// TwinCAT 3 PLC project MONETSRuntime
// Title: MONETS
// Company: IAG
// ProjectVersion: 1.2.0
// ProgramVersion: 3.1.4026.13
// libraries:
//   AstroBROT, * (BROT)
//   BROTLib, * (BROT)
//   HalfBROT, * (BROT)
//   MONET Roof, * (Georg-August-Universitaet Goettingen)
//   MONETcommon, * (IAG)
//   Tc2_DataExchange, * (Beckhoff Automation GmbH)
//   Tc2_Math, * (Beckhoff Automation GmbH)
//   Tc2_MC2, * (Beckhoff Automation GmbH)
//   Tc2_MC2_Drive, * (Beckhoff Automation GmbH)
//   Tc2_NC, * (Beckhoff Automation GmbH)
//   Tc2_Standard, * (Beckhoff Automation GmbH)
//   Tc2_System, * (Beckhoff Automation GmbH)
//   Tc2_Utilities, * (Beckhoff Automation GmbH)
//   Tc3_IotBase, * (Beckhoff Automation GmbH)
//   Tc3_JsonXml, * (Beckhoff Automation GmbH)
//   Tc3_Module, * (Beckhoff Automation GmbH)
//   VisuDialogs, * (System)
//   VisuElemEventTable, * (System)
//   VisuSymbols,3.5.10.0,System
// project tree:
//   / GlobalTextList.TcGTLO, PlcTask.TcTTO (not stored), VisualizationManager.TcVMO (not stored)
//   POUs/ FB_TelescopeAuxiliary.TcPOU, FB_WeatherCheck.TcPOU, MAIN.TcPOU
//   VISUs/ Azimuth.TcVIS, Cover.TcVIS, Derotator.TcVIS, Elevation.TcVIS, Focus.TcVIS, Hydraulics.TcVIS, Pendant.TcVIS, Safety.TcVIS, Telescope.TcVIS, Visualization.TcVIS, Roof.TcVIS
//   GVLs/ Global_Version.TcGVL
// real-time tasks:
//   TASK PlcTask: cycle T#10ms, priority 20, ADS port 350
// motion (NC):
//   TASK NC-Task 1 SAF: cycle T#2ms, priority 4, ADS port 501
//   TASK NC-Task 1 SVB: cycle T#10ms, priority 8, ADS port 511
//   AXIS Azimuth (id 1)
//     General: UnitName=°
//     Dynamic: AccelerationMaximum=10, DecelerationMaximum=10, Acceleration=3, Deceleration=3, Jerk=1
//     Velo: RefSearch=2, RefSync=2, SlowManual=1, FastManual=5, Fast=684, Maximum=10
//     OtherSettings: AllowMotionCmdToSlave=true
//     encoder EncType=8
//       EncPara: ScaleFactorNumerator=360, ScaleFactorDenominator=1048576, MaxCount=#xffffffff
//         SoftEndMinControl: Enable=true, Range=-274
//         SoftEndMaxControl: Enable=true, Range=270
//         Inc: RefMode=2
//     drive DrvType=9
//       DrvPara: MaxCount=#xffffffff, DriveControlDWord=#x00030100
//         Analog: VeloReferenz=752.4, VeloScale=1.02400649589962, TorqueSetpointScale=10, ScaleFactorActTorque=0.1
//         TimeComp: TaskDelayCycles=1
//     controller CtrType=1
//       CtrPara: PriorControlFactor=1
//         PosDiffControl: Range=10
//         Observer: BandWidth=20
//   AXIS Elevation (id 2)
//     General: UnitName=°
//     Dynamic: AccelerationMaximum=10, DecelerationMaximum=10, Acceleration=3, Deceleration=3, Jerk=2
//     Velo: RefSearch=1, RefSync=2, SlowManual=1, FastManual=3, Fast=1425, Maximum=10
//     OtherSettings: AllowMotionCmdToSlave=true
//     encoder EncType=8
//       EncPara: ScaleFactorNumerator=360, ScaleFactorDenominator=1048576, MaxCount=#xffffffff
//         SoftEndMinControl: Enable=true
//         SoftEndMaxControl: Enable=true, Range=91
//         Inc: RefMode=2
//     drive DrvType=9
//       DrvPara: MaxCount=#xffffffff, DriveControlDWord=#x00030100
//         Analog: VeloReferenz=1567.5, VeloScale=1.02400649589962, TorqueSetpointScale=10, ScaleFactorActTorque=0.1
//         TimeComp: TaskDelayCycles=1
//     controller CtrType=1
//       CtrPara: PriorControlFactor=1
//         Observer: BandWidth=20
//   AXIS Derotator (id 3)
//     General: UnitName=°
//     Dynamic: AccelerationMaximum=20, DecelerationMaximum=20, Acceleration=17.5833776855469, Deceleration=17.5833776855469, Jerk=52.7501330566406
//     Velo: RefSearch=1, RefSync=0.5, SlowManual=0.5, FastManual=5, Fast=11.7222517903646, Maximum=11.7222517903646
//     OtherSettings: AllowMotionCmdToSlave=true
//     encoder EncType=8
//       EncPara: ScaleFactorNumerator=0.2, ScaleFactorDenominator=1048576, Offset=255.939444732666, MaxCount=#xffffffff, ReferenceSystem=1
//         SoftEndMinControl: Enable=true, Range=-90
//         SoftEndMaxControl: Enable=true, Range=360
//     drive DrvType=9
//       DrvPara: MaxCount=#xffffffff, DriveControlDWord=#x00030100
//         Analog: VeloReferenz=12.894476969401, VeloScale=1.02400649589962, TorqueSetpointScale=10, ScaleFactorActTorque=0.1
//         TimeComp: TaskDelayCycles=1
//     controller CtrType=1
//       CtrPara: PriorControlFactor=1
//         Observer: BandWidth=20
//   AXIS Focus (id 4)
//     Dynamic: AccelerationMaximum=100, DecelerationMaximum=100, Acceleration=4.5, Deceleration=4.5, Jerk=13.5
//     Velo: RefSearch=0.2, RefSync=0.2, SlowManual=0.1, FastManual=0.5, Maximum=5
//     OtherSettings: AllowMotionCmdToSlave=true, PulseDistancePos=1, PulseDistanceNeg=1
//     encoder EncType=4
//       EncPara: ScaleFactorNumerator=0.001, ScaleFactorDenominator=5, Inverse=true, MaxCount=#x0000ffff
//         SoftEndMaxControl: Range=100
//         Inc: RefMode=2, RefSoftSyncMask=#x0000ffff
//     drive DrvType=23
//       DrvPara: Inverse=true
//         Analog: VeloReferenz=10.27313178, TorqueSetpointScale=10, ScaleFactorActTorque=0.1
//         TimeComp: TaskDelayCycles=1
//     controller CtrType=1
//       CtrPara: PriorControlFactor=1
//         PID: PosKp=200
//         Observer: BandWidth=20
// I/O:
//   DEVICE Device 1 (EtherCAT), AmsNetId 0.0.0.0.2.1
//     Term 8 (EK1200) [EK1200-5000 EtherCAT Power supply (2A E-Bus)]
//       Term 25 (EL1004) [EL1004 4Ch. Dig. Input 24V, 3ms]
//       Temperature IN (EL3202) [EL3202 2Ch. Ana. Input PT100 (RTD)]
//       Brake AzEl (EL2004) [EL2004 4Ch. Dig. Output 24V, 0.5A]
//       Safety Logic (EL6910) [EL6910, TwinSAFE PLC]
//       Safety IN (EL1904) [EL1904, 4 Ch. Safety Input 24V, TwinSAFE]
//         modules: Module 1 (FSOES)
//       Safety OUT (EL2904) [EL2904, 4 Ch. Safety Output 24V, 0.5A, TwinSAFE]
//         modules: Module 1 (FSOES), Module 2 (DO)
//       Hydraulics OUT (EL2008) [EL2008 8Ch. Dig. Output 24V, 0.5A]
//       Hydraulics Focus IN (EL1008) [EL1008 8Ch. Dig. Input 24V, 3ms]
//       Hydraulics IN2 (EL1008) [EL1008 8Ch. Dig. Input 24V, 3ms]
//       Focus Encoder (EL5101-0010) [EL5101-0010 1Ch. Inc. Encoder 5V (20 million increments/s)]
//       Focus Motor (EL7342) [EL7342 2Ch. DC motor output stage (50V, 3.5A)]
//       Mirror Temperature IN (EL3164) [EL3164 4Ch. Ana. Input 0-10V]
//       Power Analysis (EL3483) [EL3483 3Ch. Mains Monitoring]
//       Power (EL9410) [EL9410 E-Bus Power Supplier  (Diagnostics)]
//       Mirror Cover OUT1 (EL2004) [EL2004 4Ch. Dig. Output 24V, 0.5A]
//       Mirror Cover OUT2 (EL2004) [EL2004 4Ch. Dig. Output 24V, 0.5A]
//       Mirror Cover IN (EL1008) [EL1008 8Ch. Dig. Input 24V, 3ms]
//       Front Panel IN (EL1008) [EL1008 8Ch. Dig. Input 24V, 3ms]
//       Front Panel OUT (EL2004) [EL2004 4Ch. Dig. Output 24V, 0.5A]
//       Pendant Control IN (EL1008) [EL1008 8Ch. Dig. Input 24V, 3ms]
//       Pendant Control IN2 (EL1008) [EL1008 8Ch. Dig. Input 24V, 3ms]
//       Pendant Control OUT (EL2008) [EL2008 8Ch. Dig. Output 24V, 0.5A]
//       Cabinet OUT (EL2004) [EL2004 4Ch. Dig. Output 24V, 0.5A]
//       Term 32 (EL9011) [EL9011 End Terminal]
//   DEVICE Device 4 (EtherCAT), AmsNetId 0.0.0.0.5.1
//     Azimuth (AX5125-0000-0214) [AX5125-0000-0214 EtherCAT Drive (SoE, 1 Ch.)]
//       Term 9 (AX5805) [AX5805 (Safety Drive Option)]
//         modules: Module 1 (Safety Process Data, 1 axis), Module 2 (Standard Process Data, 1 axis)
//     Elevation (AX5125-0000-0214) [AX5125-0000-0214 EtherCAT Drive (SoE, 1 Ch.)]
//       Term 11 (AX5805) [AX5805 (Safety Drive Option)]
//         modules: Module 1 (Safety Process Data, 1 axis), Module 2 (Standard Process Data, 1 axis)
//     Derotator (AX5206-0000-0215) [AX5206-0000-0215 EtherCAT Drive (SoE, 2 Ch.)]
//       Term 13 (AX5805) [AX5805 (Safety Drive Option)]
//         modules: Module 1 (Safety Process Data, 2 axis), Module 2 (Standard Process Data, 2 axis)
//     Term 11 (EK1100) [EK1100 EtherCAT Coupler (2A E-Bus)]
//       Roof Open/Close (EL2008) [EL2008 8Ch. Dig. Output 24V, 0.5A]
//       Roof Reset (EL2008) [EL2008 8Ch. Dig. Output 24V, 0.5A]
//       Roof Safety OUT (EL2904) [EL2904, 4 Ch. Safety Output 24V, 0.5A, TwinSAFE]
//         modules: Module 1 (FSOES), Module 2 (DO)
//       Roof Safety IN (EL1904) [EL1904, 4 Ch. Safety Input 24V, TwinSAFE]
//         modules: Module 1 (FSOES)
//       Roof IN 1 (EL1008) [EL1008 8Ch. Dig. Input 24V, 3ms]
//       Roof IN 2 (EL1008) [EL1008 8Ch. Dig. Input 24V, 3ms]
//       Roof IN 3 (EL1008) [EL1008 8Ch. Dig. Input 24V, 3ms]
//       Roof Speed (EL4004) [EL4004 4Ch. Ana. Output 0-10V, 12bit]
//       Term 16 (EL9011) [EL9011 End Terminal]
// variable links:
//   Device 1 (EtherCAT) <-> Device 1 (EtherCAT)/Term 8 (EK1200)/Safety IN (EL1904)
//     Term 8 (EK1200)/Safety Logic (EL6910)/ConnectionInputs/Message_7 TxPDO <-> Module 1 (FSOES)/RxPDO/FSOE
//   Device 1 (EtherCAT) <-> Device 1 (EtherCAT)/Term 8 (EK1200)/Safety Logic (EL6910)
//     Term 8 (EK1200)/Safety IN (EL1904)/Module 1 (FSOES)/TxPDO/FSOE <-> ConnectionOutputs/Message_7 RxPDO
//     Term 8 (EK1200)/Safety OUT (EL2904)/Module 1 (FSOES)/RxPDO/FSOE <-> ConnectionInputs/Message_8 TxPDO
//   Device 1 (EtherCAT) <-> Device 1 (EtherCAT)/Term 8 (EK1200)/Safety OUT (EL2904)
//     Term 8 (EK1200)/Safety Logic (EL6910)/ConnectionOutputs/Message_8 RxPDO <-> Module 1 (FSOES)/TxPDO/FSOE
//   Device 1 (EtherCAT) <-> Device 4 (EtherCAT)/Azimuth (AX5125-0000-0214)/Term 9 (AX5805)
//     Term 8 (EK1200)/Safety Logic (EL6910)/ConnectionInputs/Message_5 TxPDO <-> Module 1 (Safety Process Data, 1 axis)/Outputs (Controlword)/FSOE
//   Device 1 (EtherCAT) <-> Device 4 (EtherCAT)/Derotator (AX5206-0000-0215)/Term 13 (AX5805)
//     Term 8 (EK1200)/Safety Logic (EL6910)/ConnectionInputs/Message_17 TxPDO <-> Module 1 (Safety Process Data, 2 axis)/Outputs (Controlword)/FSOE
//   Device 1 (EtherCAT) <-> Device 4 (EtherCAT)/Elevation (AX5125-0000-0214)/Term 11 (AX5805)
//     Term 8 (EK1200)/Safety Logic (EL6910)/ConnectionOutputs/Message_6 RxPDO <-> Module 1 (Safety Process Data, 1 axis)/Inputs (Statusword)/FSOE
//   Device 1 (EtherCAT) <-> Device 4 (EtherCAT)/Term 11 (EK1100)/Roof Safety IN (EL1904)
//     Term 8 (EK1200)/Safety Logic (EL6910)/ConnectionInputs/Message_29 TxPDO <-> Module 1 (FSOES)/RxPDO/FSOE
//   Device 1 (EtherCAT) <-> Device 4 (EtherCAT)/Term 11 (EK1100)/Roof Safety OUT (EL2904)
//     Term 8 (EK1200)/Safety Logic (EL6910)/ConnectionOutputs/Message_30 RxPDO <-> Module 1 (FSOES)/TxPDO/FSOE
//   Device 4 (EtherCAT) <-> Device 1 (EtherCAT)/Term 8 (EK1200)/Safety Logic (EL6910)
//     Azimuth (AX5125-0000-0214)/Term 9 (AX5805)/Module 1 (Safety Process Data, 1 axis)/Inputs (Statusword)/FSOE <-> ConnectionOutputs/Message_5 RxPDO
//     Derotator (AX5206-0000-0215)/Term 13 (AX5805)/Module 1 (Safety Process Data, 2 axis)/Inputs (Statusword)/FSOE <-> ConnectionOutputs/Message_17 RxPDO
//     Elevation (AX5125-0000-0214)/Term 11 (AX5805)/Module 1 (Safety Process Data, 1 axis)/Outputs (Controlword)/FSOE <-> ConnectionInputs/Message_6 TxPDO
//     Term 11 (EK1100)/Roof Safety IN (EL1904)/Module 1 (FSOES)/TxPDO/FSOE <-> ConnectionOutputs/Message_29 RxPDO
//     Term 11 (EK1100)/Roof Safety OUT (EL2904)/Module 1 (FSOES)/RxPDO/FSOE <-> ConnectionInputs/Message_30 TxPDO
//   NC-Task 1 SAF/Axes/Azimuth <-> Device 4 (EtherCAT)/Azimuth (AX5125-0000-0214)
//     Drive/Inputs/In/nDataIn1 <-> AT/Following distance
//     Drive/Inputs/In/nDataIn3[0] <-> AT/Torque/force feedback value
//     Drive/Inputs/In/nDcOutputTime <-> InfoData/DcOutputShift
//     Drive/Inputs/In/nState1 <-> AT/Drive status word @bit 8
//     Drive/Inputs/In/nState2 <-> AT/Drive status word
//     Drive/Inputs/In/nState4 @bit 1 <-> WcState/InputToggle
//     Drive/Inputs/In/nState4 <-> WcState/WcState
//     Drive/Outputs/Out/nCtrl1 <-> MDT/Master control word @bit 8
//     Drive/Outputs/Out/nDataOut1 <-> MDT/Position command value
//     Enc/Inputs/In/nDataIn1 <-> AT/Position feedback 1 value
//     Enc/Inputs/In/nDataIn3 <-> AT/Probe value 1 positive edge
//     Enc/Inputs/In/nDataIn7 <-> AT/Velocity feedback 1 value
//     Enc/Inputs/In/nDcInputTime <-> InfoData/DcInputShift
//     Enc/Inputs/In/nState4 @bit 1 <-> WcState/InputToggle
//     Enc/Inputs/In/nState4 <-> WcState/WcState
//     Enc/Inputs/In/nState5 <-> AT/Probe 1 positive latched
//     Enc/Outputs/Out/nCtrl5 <-> MDT/Probe 1 enable
//   NC-Task 1 SAF/Axes/Derotator <-> Device 4 (EtherCAT)/Derotator (AX5206-0000-0215)
//     Drive/Inputs/In/nDataIn1 <-> AT 2/Following distance
//     Drive/Inputs/In/nDataIn3[0] <-> AT 2/Torque/force feedback value
//     Drive/Inputs/In/nDcOutputTime <-> InfoData/DcOutputShift
//     Drive/Inputs/In/nState1 <-> AT 2/Drive status word @bit 8
//     Drive/Inputs/In/nState2 <-> AT 2/Drive status word
//     Drive/Inputs/In/nState4 @bit 1 <-> WcState/InputToggle
//     Drive/Inputs/In/nState4 <-> WcState/WcState
//     Drive/Outputs/Out/nCtrl1 <-> MDT 2/Master control word @bit 8
//     Drive/Outputs/Out/nDataOut1 <-> MDT 2/Position command value
//     Enc/Inputs/In/nDataIn1 <-> AT 2/Position feedback 1 value
//     Enc/Inputs/In/nDataIn7 <-> AT 2/Velocity feedback 1 value
//     Enc/Inputs/In/nDcInputTime <-> InfoData/DcInputShift
//     Enc/Inputs/In/nState4 @bit 1 <-> WcState/InputToggle
//     Enc/Inputs/In/nState4 <-> WcState/WcState
//   NC-Task 1 SAF/Axes/Elevation <-> Device 4 (EtherCAT)/Elevation (AX5125-0000-0214)
//     Drive/Inputs/In/nDataIn1 <-> AT/Following distance
//     Drive/Inputs/In/nDataIn3[0] <-> AT/Torque/force feedback value
//     Drive/Inputs/In/nDcOutputTime <-> InfoData/DcOutputShift
//     Drive/Inputs/In/nState1 <-> AT/Drive status word @bit 8
//     Drive/Inputs/In/nState2 <-> AT/Drive status word
//     Drive/Inputs/In/nState4 @bit 1 <-> WcState/InputToggle
//     Drive/Inputs/In/nState4 <-> WcState/WcState
//     Drive/Outputs/Out/nCtrl1 <-> MDT/Master control word @bit 8
//     Drive/Outputs/Out/nDataOut1 <-> MDT/Position command value
//     Enc/Inputs/In/nDataIn1 <-> AT/Position feedback 1 value
//     Enc/Inputs/In/nDataIn3 <-> AT/Probe value 1 positive edge
//     Enc/Inputs/In/nDataIn7 <-> AT/Velocity feedback 1 value
//     Enc/Inputs/In/nDcInputTime <-> InfoData/DcInputShift
//     Enc/Inputs/In/nState4 @bit 1 <-> WcState/InputToggle
//     Enc/Inputs/In/nState4 <-> WcState/WcState
//     Enc/Inputs/In/nState5 <-> AT/Probe 1 positive latched
//     Enc/Outputs/Out/nCtrl5 <-> MDT/Probe 1 enable
//   NC-Task 1 SAF/Axes/Focus <-> Device 1 (EtherCAT)/Term 8 (EK1200)/Focus Encoder (EL5101-0010)
//     Enc/Inputs/In/nDataIn1[0] <-> ENC Status compact/Counter value
//     Enc/Inputs/In/nDataIn2[0] <-> ENC Status compact/Latch value
//     Enc/Inputs/In/nState1 <-> ENC Status compact/Status/Latch C valid
//     Enc/Inputs/In/nState1 @bit 1 <-> ENC Status compact/Status/Latch extern valid
//     Enc/Inputs/In/nState1 @bit 6 <-> ENC Status compact/Status/Open circuit
//     Enc/Inputs/In/nState1 @bit 2 <-> ENC Status compact/Status/Set counter done
//     Enc/Inputs/In/nState1 @bit 5 <-> ENC Status compact/Status/Status of input status
//     Enc/Inputs/In/nState2 @bit 4 <-> ENC Status compact/Status/Status of extern latch
//     Enc/Inputs/In/nState2 <-> ENC Status compact/Status/Status of input A
//     Enc/Inputs/In/nState2 @bit 1 <-> ENC Status compact/Status/Status of input B
//     Enc/Inputs/In/nState2 @bit 2 <-> ENC Status compact/Status/Status of input C
//     Enc/Inputs/In/nState2 @bit 3 <-> ENC Status compact/Status/Status of input gate
//     Enc/Inputs/In/nState2 @bit 5 <-> ENC Status compact/Status/Sync error
//     Enc/Inputs/In/nState2 @bit 6 <-> ENC Status compact/Status/TxPDO State
//     Enc/Inputs/In/nState2 @bit 7 <-> ENC Status compact/Status/TxPDO Toggle
//     Enc/Inputs/In/nState4 @bit 1 <-> WcState/InputToggle
//     Enc/Inputs/In/nState4 <-> WcState/WcState
//     Enc/Outputs/Out/nCtrl1 <-> ENC Control compact/Control/Enable latch C
//     Enc/Outputs/Out/nCtrl1 @bit 3 <-> ENC Control compact/Control/Enable latch extern on negative edge
//     Enc/Outputs/Out/nCtrl1 @bit 1 <-> ENC Control compact/Control/Enable latch extern on positive edge
//     Enc/Outputs/Out/nCtrl1 @bit 2 <-> ENC Control compact/Control/Set counter
//     Enc/Outputs/Out/nDataOut1[0] <-> ENC Control compact/Set counter value
//   NC-Task 1 SAF/Axes/Focus <-> Device 1 (EtherCAT)/Term 8 (EK1200)/Focus Motor (EL7342)
//     Drive/Inputs/In/nState1 @bit 3 <-> DCM Status Channel 1/Status/Error
//     Drive/Inputs/In/nState1 @bit 5 <-> DCM Status Channel 1/Status/Moving negative
//     Drive/Inputs/In/nState1 @bit 4 <-> DCM Status Channel 1/Status/Moving positive
//     Drive/Inputs/In/nState1 @bit 1 <-> DCM Status Channel 1/Status/Ready
//     Drive/Inputs/In/nState1 <-> DCM Status Channel 1/Status/Ready to enable
//     Drive/Inputs/In/nState1 @bit 6 <-> DCM Status Channel 1/Status/Torque reduced
//     Drive/Inputs/In/nState1 @bit 2 <-> DCM Status Channel 1/Status/Warning
//     Drive/Inputs/In/nState2 @bit 3 <-> DCM Status Channel 1/Status/Digital input 1
//     Drive/Inputs/In/nState2 @bit 4 <-> DCM Status Channel 1/Status/Digital input 2
//     Drive/Inputs/In/nState2 @bit 5 <-> DCM Status Channel 1/Status/Sync error
//     Drive/Inputs/In/nState2 @bit 7 <-> DCM Status Channel 1/Status/TxPDO Toggle
//     Drive/Inputs/In/nState4 @bit 1 <-> WcState/InputToggle
//     Drive/Inputs/In/nState4 <-> WcState/WcState
//     Drive/Outputs/Out/nCtrl1 <-> DCM Control Channel 1/Control/Enable
//     Drive/Outputs/Out/nCtrl1 @bit 2 <-> DCM Control Channel 1/Control/Reduce torque
//     Drive/Outputs/Out/nCtrl1 @bit 1 <-> DCM Control Channel 1/Control/Reset
//     Drive/Outputs/Out/nCtrl1 @bit 3 <-> DCM Control Channel 1/Control/Threshold active
//     Drive/Outputs/Out/nDataOut2[0] <-> DCM Velocity Channel 1/Velocity
//   MONETSRuntime/MONETSRuntime Instance <-> Device 1 (EtherCAT)/Term 8 (EK1200)/Brake AzEl (EL2004)
//     PlcTask Outputs/MAIN.HydraulicsControl.ObBrakeAzEl <-> Channel 2/MAIN.HydraulicsControl.ObBrakeAzEl
//   MONETSRuntime/MONETSRuntime Instance <-> Device 1 (EtherCAT)/Term 8 (EK1200)/Front Panel IN (EL1008)
//     PlcTask Inputs/MAIN.CabinetControl.inButtonReset <-> Channel 3/MAIN.CabinetControl.inButtonReset
//     PlcTask Inputs/MAIN.CabinetControl.inButtonStart <-> Channel 1/MAIN.CabinetControl.inButtonStart
//     PlcTask Inputs/MAIN.CabinetControl.inButtonStop <-> Channel 2/MAIN.CabinetControl.inButtonStop
//     PlcTask Inputs/MAIN.CabinetControl.inKeyClearBrakes <-> Channel 5/MAIN.CabinetControl.inKeyClearBrakes
//     PlcTask Inputs/MAIN.CabinetControl.inKeyLocal <-> Channel 4/MAIN.CabinetControl.inKeyLocal
//   MONETSRuntime/MONETSRuntime Instance <-> Device 1 (EtherCAT)/Term 8 (EK1200)/Front Panel OUT (EL2004)
//     PlcTask Outputs/MAIN.CabinetControl.outLampError <-> Channel 3/MAIN.CabinetControl.outLampError
//     PlcTask Outputs/MAIN.CabinetControl.outLampManual <-> Channel 2/MAIN.CabinetControl.outLampManual
//     PlcTask Outputs/MAIN.CabinetControl.outLampPower <-> Channel 1/MAIN.CabinetControl.outLampPower
//   MONETSRuntime/MONETSRuntime Instance <-> Device 1 (EtherCAT)/Term 8 (EK1200)/Hydraulics Focus IN (EL1008)
//     PlcTask Inputs/MAIN.FocusControl.IbLimitFar <-> Channel 5/MAIN.FocusControl.IbLimitFar
//     PlcTask Inputs/MAIN.FocusControl.IbLimitNear <-> Channel 4/MAIN.FocusControl.IbLimitNear
//     PlcTask Inputs/MAIN.HydraulicsControl.IbPumpRunning <-> Channel 1/MAIN.HydraulicsControl.IbPumpRunning
//     PlcTask Inputs/MAIN.HydraulicsControl.IbSuctionRunning <-> Channel 2/MAIN.HydraulicsControl.IbSuctionRunning
//   MONETSRuntime/MONETSRuntime Instance <-> Device 1 (EtherCAT)/Term 8 (EK1200)/Hydraulics IN2 (EL1008)
//     PlcTask Inputs/MAIN.HydraulicsControl.IbOilCold <-> Channel 5/MAIN.HydraulicsControl.IbOilCold
//     PlcTask Inputs/MAIN.HydraulicsControl.IbOilFilterDirty <-> Channel 6/MAIN.HydraulicsControl.IbOilFilterDirty
//     PlcTask Inputs/MAIN.HydraulicsControl.IbOilHigh <-> Channel 2/MAIN.HydraulicsControl.IbOilHigh
//     PlcTask Inputs/MAIN.HydraulicsControl.IbOilHot <-> Channel 4/MAIN.HydraulicsControl.IbOilHot
//     PlcTask Inputs/MAIN.HydraulicsControl.IbOilLow <-> Channel 1/MAIN.HydraulicsControl.IbOilLow
//     PlcTask Inputs/MAIN.HydraulicsControl.IbOilPressureOK <-> Channel 3/MAIN.HydraulicsControl.IbOilPressureOK
//     PlcTask Inputs/MAIN.HydraulicsControl.IbOilReserve <-> Channel 8/MAIN.HydraulicsControl.IbOilReserve
//     PlcTask Inputs/MAIN.HydraulicsControl.IbOilpanMaximum <-> Channel 7/MAIN.HydraulicsControl.IbOilpanMaximum
//   MONETSRuntime/MONETSRuntime Instance <-> Device 1 (EtherCAT)/Term 8 (EK1200)/Hydraulics OUT (EL2008)
//     PlcTask Outputs/MAIN.FocusControl.ObFocusUnlock <-> Channel 7/MAIN.FocusControl.ObFocusUnlock
//     PlcTask Outputs/MAIN.HydraulicsControl.ObOilPumpEnable <-> Channel 1/MAIN.HydraulicsControl.ObOilPumpEnable
//     PlcTask Outputs/MAIN.HydraulicsControl.ObOilSuctionEnable <-> Channel 3/MAIN.HydraulicsControl.ObOilSuctionEnable
//     PlcTask Outputs/MAIN.HydraulicsControl.ObResetOilPump <-> Channel 2/MAIN.HydraulicsControl.ObResetOilPump
//     PlcTask Outputs/MAIN.HydraulicsControl.ObResetSuctionPump <-> Channel 4/MAIN.HydraulicsControl.ObResetSuctionPump
//   MONETSRuntime/MONETSRuntime Instance <-> Device 1 (EtherCAT)/Term 8 (EK1200)/Mirror Cover IN (EL1008)
//     PlcTask Inputs/MAIN.CoverControl.IabCoverClosed[1] <-> Channel 2/MAIN.CoverControl.IabCoverClosed[1]
//     PlcTask Inputs/MAIN.CoverControl.IabCoverClosed[2] <-> Channel 4/MAIN.CoverControl.IabCoverClosed[2]
//     PlcTask Inputs/MAIN.CoverControl.IabCoverClosed[3] <-> Channel 6/MAIN.CoverControl.IabCoverClosed[3]
//     PlcTask Inputs/MAIN.CoverControl.IabCoverOpen[1] <-> Channel 1/MAIN.CoverControl.IabCoverOpen[1]
//     PlcTask Inputs/MAIN.CoverControl.IabCoverOpen[2] <-> Channel 3/MAIN.CoverControl.IabCoverOpen[2]
//     PlcTask Inputs/MAIN.CoverControl.IabCoverOpen[3] <-> Channel 5/MAIN.CoverControl.IabCoverOpen[3]
//   MONETSRuntime/MONETSRuntime Instance <-> Device 1 (EtherCAT)/Term 8 (EK1200)/Mirror Cover OUT1 (EL2004)
//     PlcTask Outputs/MAIN.CoverControl.OabCloseCover[1] <-> Channel 2/MAIN.CoverControl.OabCloseCover[1]
//     PlcTask Outputs/MAIN.CoverControl.OabCloseCover[2] <-> Channel 4/MAIN.CoverControl.OabCloseCover[2]
//     PlcTask Outputs/MAIN.CoverControl.OabOpenCover[1] <-> Channel 1/MAIN.CoverControl.OabOpenCover[1]
//     PlcTask Outputs/MAIN.CoverControl.OabOpenCover[2] <-> Channel 3/MAIN.CoverControl.OabOpenCover[2]
//   MONETSRuntime/MONETSRuntime Instance <-> Device 1 (EtherCAT)/Term 8 (EK1200)/Mirror Cover OUT2 (EL2004)
//     PlcTask Outputs/MAIN.CoverControl.OabCloseCover[3] <-> Channel 2/MAIN.CoverControl.OabCloseCover[3]
//     PlcTask Outputs/MAIN.CoverControl.OabOpenCover[3] <-> Channel 1/MAIN.CoverControl.OabOpenCover[3]
//   MONETSRuntime/MONETSRuntime Instance <-> Device 1 (EtherCAT)/Term 8 (EK1200)/Mirror Temperature IN (EL3164)
//     PlcTask Inputs/MAIN.HydraulicsControl.InOilLevel <-> OilLevel/MAIN.HydraulicsControl.InOilLevel
//     PlcTask Inputs/MAIN.TelescopeAuxiliary.tempSensorFlange <-> AI Standard Channel 2/MAIN.TelescopeAuxiliary.tempSensorFlange
//     PlcTask Inputs/MAIN.TelescopeAuxiliary.tempSensorM1 <-> AI Standard Channel 4/MAIN.TelescopeAuxiliary.tempSensorM1
//     PlcTask Inputs/MAIN.TelescopeAuxiliary.tempSensorM2 <-> AI Standard Channel 1/MAIN.TelescopeAuxiliary.tempSensorM2
//   MONETSRuntime/MONETSRuntime Instance <-> Device 1 (EtherCAT)/Term 8 (EK1200)/Pendant Control IN (EL1008)
//     PlcTask Inputs/MAIN.PendantControl.IbBCD0 <-> Channel 1/MAIN.PendantControl.IbBCD0
//     PlcTask Inputs/MAIN.PendantControl.IbBCD2 <-> Channel 2/MAIN.PendantControl.IbBCD2
//     PlcTask Inputs/MAIN.PendantControl.IbBCD4 <-> Channel 3/MAIN.PendantControl.IbBCD4
//     PlcTask Inputs/MAIN.PendantControl.IbBCD8 <-> Channel 4/MAIN.PendantControl.IbBCD8
//     PlcTask Inputs/MAIN.PendantControl.IbDirectionDown <-> Channel 7/MAIN.PendantControl.IbDirectionDown
//     PlcTask Inputs/MAIN.PendantControl.IbDirectionUp <-> Channel 6/MAIN.PendantControl.IbDirectionUp
//     PlcTask Inputs/MAIN.PendantControl.IbEnableKey <-> Channel 8/MAIN.PendantControl.IbEnableKey
//     PlcTask Inputs/MAIN.PendantControl.IbResetButton <-> Channel 5/MAIN.PendantControl.IbResetButton
//   MONETSRuntime/MONETSRuntime Instance <-> Device 1 (EtherCAT)/Term 8 (EK1200)/Pendant Control IN2 (EL1008)
//     PlcTask Inputs/MAIN.PendantControl.IbDirectionLeft <-> Channel 2/MAIN.PendantControl.IbDirectionLeft
//     PlcTask Inputs/MAIN.PendantControl.IbDirectionRight <-> Channel 3/MAIN.PendantControl.IbDirectionRight
//     PlcTask Inputs/MAIN.PendantControl.IbEnableButton <-> Channel 1/MAIN.PendantControl.IbEnableButton
//   MONETSRuntime/MONETSRuntime Instance <-> Device 1 (EtherCAT)/Term 8 (EK1200)/Pendant Control OUT (EL2008)
//     PlcTask Outputs/MAIN.PendantControl.ObLampDown <-> Channel 2/MAIN.PendantControl.ObLampDown
//     PlcTask Outputs/MAIN.PendantControl.ObLampError <-> Channel 5/MAIN.PendantControl.ObLampError
//     PlcTask Outputs/MAIN.PendantControl.ObLampLeft <-> Channel 4/MAIN.PendantControl.ObLampLeft
//     PlcTask Outputs/MAIN.PendantControl.ObLampRight <-> Channel 3/MAIN.PendantControl.ObLampRight
//     PlcTask Outputs/MAIN.PendantControl.ObLampUp <-> Channel 1/MAIN.PendantControl.ObLampUp
//   MONETSRuntime/MONETSRuntime Instance <-> Device 1 (EtherCAT)/Term 8 (EK1200)/Power Analysis (EL3483)
//     PlcTask Inputs/MAIN.PowerMonitoring.FrequencyGuardError <-> Total Status/Frequency Guard Error
//     PlcTask Inputs/MAIN.PowerMonitoring.FrequencyGuardWarning <-> Total Status/Frequency Guard Warning
//     PlcTask Inputs/MAIN.PowerMonitoring.L1InaccVoltage <-> L1 Status/Inaccurate Voltage
//     PlcTask Inputs/MAIN.PowerMonitoring.L2InaccVoltage <-> L2 Status/Inaccurate Voltage
//     PlcTask Inputs/MAIN.PowerMonitoring.L3InaccVoltage <-> L3 Status/Inaccurate Voltage
//     PlcTask Inputs/MAIN.PowerMonitoring.L1OverVoltage <-> L1 Status/Voltage Guard Warning
//     PlcTask Inputs/MAIN.PowerMonitoring.L1VoltageGuardError <-> L1 Status/Voltage Guard Error
//     PlcTask Inputs/MAIN.PowerMonitoring.L2VoltageGuardError <-> L2 Status/Voltage Guard Error
//     PlcTask Inputs/MAIN.PowerMonitoring.L3VoltageGuardError <-> L3 Status/Voltage Guard Error
//     PlcTask Inputs/MAIN.PowerMonitoring.L1VoltageGuardWarning <-> L1 Status/Voltage Guard Warning
//     PlcTask Inputs/MAIN.PowerMonitoring.L2VoltageGuardWarning <-> L2 Status/Voltage Guard Warning
//     PlcTask Inputs/MAIN.PowerMonitoring.L3VoltageGuardWarning <-> L3 Status/Voltage Guard Warning
//     PlcTask Inputs/MAIN.PowerMonitoring.L2OverVoltage <-> L2 Status/Overvoltage
//     PlcTask Inputs/MAIN.PowerMonitoring.L3OverVoltage <-> L3 Status/Overvoltage
//     PlcTask Inputs/MAIN.PowerMonitoring.PowerQuality <-> Total Status/Power Quality Factor
//     PlcTask Inputs/MAIN.PowerMonitoring.QualityGuardError <-> Total Status/Power Quality Guard Error
//     PlcTask Inputs/MAIN.PowerMonitoring.QualityGuardWarning <-> Total Status/Power Quality Guard Warning
//     PlcTask Inputs/MAIN.PowerMonitoring.UnbalanceGuardError <-> Total Advanced/Unbalance Guard Error
//     PlcTask Inputs/MAIN.PowerMonitoring.UnbalanceGuardWarning <-> Total Advanced/Unbalance Guard Warning
//   MONETSRuntime/MONETSRuntime Instance <-> Device 1 (EtherCAT)/Term 8 (EK1200)/Safety Logic (EL6910)
//     PlcTask Inputs/MAIN.AzimuthControl.IbSTO <-> StandardInputs/Standard Out Var 18
//     PlcTask Inputs/MAIN.DerotatorControl.IbSTO <-> StandardInputs/Standard Out Var 20
//     PlcTask Inputs/MAIN.ElevationControl.IbSTO <-> StandardInputs/Standard Out Var 19
//     PlcTask Inputs/MAIN.SafetyHandling.stInfoEStop1 <-> Function Block Info Data/TwinSafeGroup1.Network1.FBEstop1 Info Data
//     PlcTask Inputs/MAIN.SafetyHandling.stInfoGroup1 <-> TwinSAFE Group Info Data/TwinSafeGroup1 Info Data
//     PlcTask Inputs/MAIN.SafetyHandling.stInfoSafetyIn <-> Connection Info Data/Message_7 Info Data
//     PlcTask Inputs/MAIN.SafetyHandling.stInfoSafetyOut <-> Connection Info Data/Message_8 Info Data
//     PlcTask Outputs/MAIN.SafetyHandling.outErrAck <-> StandardOutputs/Standard In Var 1
//     PlcTask Outputs/MAIN.SafetyHandling.outResetAzimuthSTO <-> StandardOutputs/Standard In Var 25
//     PlcTask Outputs/MAIN.SafetyHandling.outResetDerotatorSTO <-> StandardOutputs/Standard In Var 22
//     PlcTask Outputs/MAIN.SafetyHandling.outResetElevationSTO <-> StandardOutputs/Standard In Var 26
//     PlcTask Outputs/MAIN.SafetyHandling.outRestart <-> StandardOutputs/Standard In Var 3
//     PlcTask Outputs/MAIN.SafetyHandling.outRun <-> StandardOutputs/Standard In Var 2
//   MONETSRuntime/MONETSRuntime Instance <-> Device 1 (EtherCAT)/Term 8 (EK1200)/Temperature IN (EL3202)
//     PlcTask Inputs/MAIN.CabinetControl.inCabinetTemp <-> RTD Inputs Channel 1/MAIN.CabinetControl.inCabinetTemp
//   MONETSRuntime/MONETSRuntime Instance <-> Device 4 (EtherCAT)/Azimuth (AX5125-0000-0214)
//     PlcTask Inputs/MAIN.AzimuthControl.InDiagnostic <-> AT/Diagnostic number
//     PlcTask Inputs/MAIN.AzimuthControl.InDigitalInputs <-> AT/Digital inputs, state
//     PlcTask Inputs/MAIN.AzimuthControl.InTorque <-> AT/Torque/force feedback value
//   MONETSRuntime/MONETSRuntime Instance <-> Device 4 (EtherCAT)/Derotator (AX5206-0000-0215)
//     PlcTask Inputs/MAIN.DerotatorControl.InDiagnostic <-> AT 1/Diagnostic number
//     PlcTask Inputs/MAIN.DerotatorControl.InDigitalInputs <-> AT 1/Digital inputs, state
//     PlcTask Inputs/MAIN.DerotatorControl.InTorque <-> AT 1/Torque/force feedback value
//   MONETSRuntime/MONETSRuntime Instance <-> Device 4 (EtherCAT)/Elevation (AX5125-0000-0214)
//     PlcTask Inputs/MAIN.ElevationControl.InDiagnostic <-> AT/Diagnostic number
//     PlcTask Inputs/MAIN.ElevationControl.InDigitalInputs <-> AT/Digital inputs, state
//     PlcTask Inputs/MAIN.ElevationControl.InTorque <-> AT/Torque/force feedback value
//   MONETSRuntime/MONETSRuntime Instance <-> Device 4 (EtherCAT)/Term 11 (EK1100)/Roof IN 1 (EL1008)
//     PlcTask Inputs/MAIN.RoofControl.automatic <-> Channel 6/MAIN.RoofControl.automatic
//     PlcTask Inputs/MAIN.RoofControl.roofs[1].motors[1].counter <-> Channel 1/MAIN.RoofControl.roofs[1].motors[1].counter
//     PlcTask Inputs/MAIN.RoofControl.roofs[1].motors[2].counter <-> Channel 7/MAIN.RoofControl.roofs[1].motors[2].counter
//     PlcTask Inputs/MAIN.RoofControl.roofs[2].motors[1].counter <-> Channel 3/MAIN.RoofControl.roofs[2].motors[1].counter
//     PlcTask Inputs/MAIN.RoofControl.roofs[2].motors[2].counter <-> Channel 5/MAIN.RoofControl.roofs[2].motors[2].counter
//     PlcTask Inputs/MAIN.RoofControl.roofs[1].motors[1].motor_error <-> Channel 2/MAIN.RoofControl.roofs[1].motors[1].motor_error
//     PlcTask Inputs/MAIN.RoofControl.roofs[2].motors[1].motor_error <-> Channel 4/MAIN.RoofControl.roofs[2].motors[1].motor_error
//     PlcTask Inputs/MAIN.RoofControl.roofs[1].open_roof <-> Channel 8/MAIN.RoofControl.roofs[1].open_roof
//   MONETSRuntime/MONETSRuntime Instance <-> Device 4 (EtherCAT)/Term 11 (EK1100)/Roof IN 2 (EL1008)
//     PlcTask Inputs/MAIN.RoofControl.roofs[1].close_roof <-> Channel 1/MAIN.RoofControl.roofs[1].close_roof
//     PlcTask Inputs/MAIN.RoofControl.roofs[2].close_roof <-> Channel 5/MAIN.RoofControl.roofs[2].close_roof
//     PlcTask Inputs/MAIN.RoofControl.roofs[1].motors[1].closed <-> Channel 6/MAIN.RoofControl.roofs[1].motors[1].closed
//     PlcTask Inputs/MAIN.RoofControl.roofs[1].motors[1].opened <-> Channel 4/MAIN.RoofControl.roofs[1].motors[1].opened
//     PlcTask Inputs/MAIN.RoofControl.roofs[2].motors[1].opened <-> Channel 8/MAIN.RoofControl.roofs[2].motors[1].opened
//     PlcTask Inputs/MAIN.RoofControl.roofs[1].motors[2].motor_error <-> Channel 2/MAIN.RoofControl.roofs[1].motors[2].motor_error
//     PlcTask Inputs/MAIN.RoofControl.roofs[2].motors[2].motor_error <-> Channel 7/MAIN.RoofControl.roofs[2].motors[2].motor_error
//     PlcTask Inputs/MAIN.RoofControl.roofs[2].open_roof <-> Channel 3/MAIN.RoofControl.roofs[2].open_roof
//   MONETSRuntime/MONETSRuntime Instance <-> Device 4 (EtherCAT)/Term 11 (EK1100)/Roof IN 3 (EL1008)
//     PlcTask Inputs/MAIN.RoofControl.roofs[1].motors[2].closed <-> Channel 2/MAIN.RoofControl.roofs[1].motors[2].closed
//     PlcTask Inputs/MAIN.RoofControl.roofs[2].motors[1].closed <-> Channel 1/MAIN.RoofControl.roofs[2].motors[1].closed
//     PlcTask Inputs/MAIN.RoofControl.roofs[2].motors[2].closed <-> Channel 5/MAIN.RoofControl.roofs[2].motors[2].closed
//     PlcTask Inputs/MAIN.RoofControl.roofs[1].motors[2].opened <-> Channel 7/MAIN.RoofControl.roofs[1].motors[2].opened
//     PlcTask Inputs/MAIN.RoofControl.roofs[2].motors[2].opened <-> Channel 3/MAIN.RoofControl.roofs[2].motors[2].opened
//   MONETSRuntime/MONETSRuntime Instance <-> Device 4 (EtherCAT)/Term 11 (EK1100)/Roof Open/Close (EL2008)
//     PlcTask Outputs/MAIN.RoofControl.roofs[1].motors[1].direction_close <-> Channel 3/MAIN.RoofControl.roofs[1].motors[1].direction_close
//     PlcTask Outputs/MAIN.RoofControl.roofs[1].motors[2].direction_close <-> Channel 8/MAIN.RoofControl.roofs[1].motors[2].direction_close
//     PlcTask Outputs/MAIN.RoofControl.roofs[2].motors[1].direction_close <-> Channel 7/MAIN.RoofControl.roofs[2].motors[1].direction_close
//     PlcTask Outputs/MAIN.RoofControl.roofs[2].motors[2].direction_close <-> Channel 4/MAIN.RoofControl.roofs[2].motors[2].direction_close
//     PlcTask Outputs/MAIN.RoofControl.roofs[1].motors[1].direction_open <-> Channel 1/MAIN.RoofControl.roofs[1].motors[1].direction_open
//     PlcTask Outputs/MAIN.RoofControl.roofs[1].motors[2].direction_open <-> Channel 6/MAIN.RoofControl.roofs[1].motors[2].direction_open
//     PlcTask Outputs/MAIN.RoofControl.roofs[2].motors[1].direction_open <-> Channel 5/MAIN.RoofControl.roofs[2].motors[1].direction_open
//     PlcTask Outputs/MAIN.RoofControl.roofs[2].motors[2].direction_open <-> Channel 2/MAIN.RoofControl.roofs[2].motors[2].direction_open
//   MONETSRuntime/MONETSRuntime Instance <-> Device 4 (EtherCAT)/Term 11 (EK1100)/Roof Reset (EL2008)
//     PlcTask Outputs/MAIN.RoofControl.roofs[1].motors[1].reset_drive <-> Channel 1/MAIN.RoofControl.roofs[1].motors[1].reset_drive
//     PlcTask Outputs/MAIN.RoofControl.roofs[1].motors[2].reset_drive <-> Channel 7/MAIN.RoofControl.roofs[1].motors[2].reset_drive
//     PlcTask Outputs/MAIN.RoofControl.roofs[2].motors[1].reset_drive <-> Channel 3/MAIN.RoofControl.roofs[2].motors[1].reset_drive
//     PlcTask Outputs/MAIN.RoofControl.roofs[2].motors[2].reset_drive <-> Channel 5/MAIN.RoofControl.roofs[2].motors[2].reset_drive
//   MONETSRuntime/MONETSRuntime Instance <-> Device 4 (EtherCAT)/Term 11 (EK1100)/Roof Speed (EL4004)
//     PlcTask Outputs/MAIN.RoofControl.roofs[1].motors[1].speed <-> AO Outputs Channel 1/MAIN.RoofControl.roofs[1].motors[1].speed
//     PlcTask Outputs/MAIN.RoofControl.roofs[1].motors[2].speed <-> AO Outputs Channel 4/MAIN.RoofControl.roofs[1].motors[2].speed
//     PlcTask Outputs/MAIN.RoofControl.roofs[2].motors[1].speed <-> AO Outputs Channel 2/MAIN.RoofControl.roofs[2].motors[1].speed
//     PlcTask Outputs/MAIN.RoofControl.roofs[2].motors[2].speed <-> AO Outputs Channel 3/MAIN.RoofControl.roofs[2].motors[2].speed
//   MONETSRuntime/MONETSRuntime Instance <-> NC-Task 1 SAF/Axes/Azimuth
//     PlcTask Inputs/MAIN.AzimuthControl.axisRef.NcToPlc <-> Outputs/ToPlc
//     PlcTask Outputs/MAIN.AzimuthControl.axisRef.PlcToNc <-> Inputs/FromPlc
//   MONETSRuntime/MONETSRuntime Instance <-> NC-Task 1 SAF/Axes/Derotator
//     PlcTask Inputs/MAIN.DerotatorControl.axisRef.NcToPlc <-> Outputs/ToPlc
//     PlcTask Outputs/MAIN.DerotatorControl.axisRef.PlcToNc <-> Inputs/FromPlc
//   MONETSRuntime/MONETSRuntime Instance <-> NC-Task 1 SAF/Axes/Elevation
//     PlcTask Inputs/MAIN.ElevationControl.axisRef.NcToPlc <-> Outputs/ToPlc
//     PlcTask Outputs/MAIN.ElevationControl.axisRef.PlcToNc <-> Inputs/FromPlc
//   MONETSRuntime/MONETSRuntime Instance <-> NC-Task 1 SAF/Axes/Focus
//     PlcTask Inputs/MAIN.FocusControl.refAxis.NcToPlc <-> Outputs/ToPlc
//     PlcTask Outputs/MAIN.FocusControl.refAxis.PlcToNc <-> Inputs/FromPlc

// ---- GVLs/Global_Version.TcGVL
{attribute 'qualified_only'}
VAR_GLOBAL CONSTANT
	// Mirrors Beckhoff's own Global_Version.stLibVersion_* pattern (see ST_LibVersion),
	// which only covers Tc2_*/Tc3_* library references, not custom ones -- until now: this
	// GVL uses Beckhoff's own naming exactly, so it merges into a consumer's Global_Version.
	// Kept in sync with <ProjectVersion> in MONETSRuntime.plcproj at release time.
	// SA0033 (unused variable) is a hard error in this project; this constant is meant
	// to be read externally via ADS, never referenced internally, so it's suppressed here.
	{attribute 'analysis' := '-33'}
	stLibVersion_MONETSRuntime : ST_LibVersion := (
		iMajor := 1,
		iMinor := 2,
		iBuild := 0,
		iRevision := 0,
		nFlags := 1,
		sVersion := '1.2.0'
	);
END_VAR

// ---- POUs/FB_TelescopeAuxiliary.TcPOU
FUNCTION_BLOCK FB_TelescopeAuxiliary
VAR
	tempSensorM1   		AT%I*: INT;
	tempSensorM1cell	AT%I*: INT;
	tempSensorM2   		AT%I*: INT;
	tempSensorFlange	AT%I*: INT;
	fbComm				: I_Comm;
END_VAR
VAR_OUTPUT
	tempM1				: REAL;
	tempM1cell			: REAL;
	tempM2				: REAL;
	tempFlange			: REAL;
END_VAR

tempM1 		:= tempSensorM1 / 32767.0 * 150.0 - 50.0; 
tempM1cell 	:= tempSensorM1cell / 32767.0 * 150.0 - 50.0;
tempM2 		:= tempSensorM2 / 32767.0 * 150.0 - 50.0;
tempFlange 	:= tempSensorFlange / 32767.0 * 150.0 - 50.0;

//FB_Init is always available implicitly and it is used primarily for initialization.
//The return value is not evaluated. For a specific influence, you can also declare the
//methods explicitly and provide additional code there with the standard initialization
//code. You can evaluate the return value.
METHOD FB_Init: BOOL
VAR_INPUT
    bInitRetains	: BOOL; // TRUE: the retain variables are initialized (reset warm / reset cold)
    bInCopyCode		: BOOL;  // TRUE: the instance will be copied to the copy code afterward (online change)
	comm			: I_Comm;	   
END_VAR
THIS^.fbComm := comm;
END_METHOD

METHOD SendTelemetry : BOOL
VAR_INPUT
END_VAR
fbComm.Publish('telescope', 'dome', 'AUXILIARY.SENSOR[1].NAME', 'TEMP_M1');
fbComm.Publish('telescope', 'dome', 'AUXILIARY.SENSOR[1].VALUE', LREAL_TO_FMTSTR(tempM1, 2, TRUE));
fbComm.Publish('telescope', 'dome', 'AUXILIARY.SENSOR[1].UNIT', 'C');
fbComm.Publish('telescope', 'dome', 'AUXILIARY.SENSOR[2].NAME', 'TEMP_M2');
fbComm.Publish('telescope', 'dome', 'AUXILIARY.SENSOR[2].VALUE', LREAL_TO_FMTSTR(tempM2, 2, TRUE));
fbComm.Publish('telescope', 'dome', 'AUXILIARY.SENSOR[2].UNIT', 'C');
fbComm.Publish('telescope', 'dome', 'AUXILIARY.SENSOR[3].NAME', 'TEMP_M1_CELL');
fbComm.Publish('telescope', 'dome', 'AUXILIARY.SENSOR[3].VALUE', LREAL_TO_FMTSTR(tempM1cell, 2, TRUE));
fbComm.Publish('telescope', 'dome', 'AUXILIARY.SENSOR[3].UNIT', 'C');
fbComm.Publish('telescope', 'dome', 'AUXILIARY.SENSOR[4].NAME', 'TEMP_FLANGE');
fbComm.Publish('telescope', 'dome', 'AUXILIARY.SENSOR[4].VALUE', LREAL_TO_FMTSTR(tempFlange, 2, TRUE));
fbComm.Publish('telescope', 'dome', 'AUXILIARY.SENSOR[4].UNIT', 'C');
END_METHOD

END_FUNCTION_BLOCK

// ---- POUs/FB_WeatherCheck.TcPOU
FUNCTION_BLOCK FB_WeatherCheck
VAR_INPUT
	bEnable				: BOOL := TRUE;
	sHostName			: STRING;
	nHostPort			: UINT;
	sUri				: STRING;
	PT					: TIME := T#10S; 
END_VAR
VAR_OUTPUT
	bBusy				: BOOL;
	bError				: BOOL;
	bWeatherGood		: BOOL;
END_VAR
VAR
	fbClient			: FB_IotHttpClient :=();
	fbRequest			: FB_IotHttpRequest;
	fbJson				: FB_JsonDomParser;
	nState				: UDINT;
	
	bGetContentResult	: BOOL;
	sContent			: STRING(511);
	
	bGetJsonResult		: BOOL;
	jsonDoc				: SJsonValue;
	jsonGood			: SJsonValue;
	
	fbTON				: TON();
END_VAR

IF NOT bEnable THEN
	RETURN;
END_IF

fbClient.Execute();

CASE nState OF
0:	
	IF NOT fbClient.bConfigured THEN
		fbClient.sHostName := sHostName;
		fbClient.nHostPort := nHostPort; 
		fbClient.bKeepAlive := TRUE;
		fbClient.tConnectionTimeout := T#10S;
	ELSE
		nState := 1;
	END_IF
1:
	IF fbRequest.SendRequest(sUri := sUri, fbClient := fbClient, eRequestType := ETcIotHttpRequestType.HTTP_GET, 0 ,0, 0) THEN				
		nState := 2;
		bBusy := TRUE;
		bError := FALSE;
	END_IF					
2:
	IF NOT fbRequest.bBusy THEN
		bError := TRUE;
		IF NOT fbRequest.bError THEN				 
			bGetContentResult := fbRequest.GetContent(pContent := ADR(sContent), nContentSize := SIZEOF(sContent), bSetNullTermination := TRUE);
			IF fbRequest.nStatusCode >= 200 AND fbRequest.nStatusCode < 300 THEN
				bGetJsonResult := FALSE;
				jsonDoc := fbRequest.GetJsonDomContent(fbJson);
				IF jsonDoc <> 0 THEN
					IF fbJson.HasMember(jsonDoc, 'good')  THEN
						jsonGood := fbJson.FindMember(jsonDoc, 'good');
						bError := FALSE;						
						IF fbJson.IsBool(jsonGood) THEN						
							bWeatherGood := fbJson.GetBool(jsonGood);
						END_IF		
					END_IF
					bError := FALSE;	
				END_IF							
			END_IF
		END_IF
		nState := 3;
		bBusy := FALSE;
	END_IF
3:
	fbTON(IN := TRUE, PT := PT);
	IF fbTON.Q THEN
		fbTON(IN := FALSE);
    	nState := 0;
	END_IF  	

END_CASE

END_FUNCTION_BLOCK

// ---- POUs/MAIN.TcPOU
PROGRAM MAIN
VAR
	ready				: BOOL;		// telescope drives are ready to enable
	error				: BOOL;
	brakeClearing		: BOOL := FALSE;	//	open brake
	
	commTimer 			: TON := (PT:=T#5S);
	getHostName			: FB_GetHostName;
	hostName			: STRING(255);
	executeHostName		: BOOL := TRUE;
	
	eTelescopeMode 		: E_TelescopeMode;
	
	fbComm				: FB_Comm_MQTT_Influx;
	SafetyHandling		: FB_MonetSafetyHandling(comm := fbComm);
	CabinetControl		: FB_MonetCabinetControl(comm := fbComm);
	PowerMonitoring		: FB_MonetPowerMonitoring(comm := fbComm);
	RoofControl			: FB_RoofControl(comm := fbComm);
	CoverControl		: FB_MonetCoverControl(comm := fbComm);
	HydraulicsControl	: FB_HydraulicsControl(comm := fbComm);
	FocusControl		: FB_FocusControl(comm := fbComm);
	DerotatorControl	: FB_DerotatorControl(comm := fbComm);
	ElevationControl	: FB_ElevationControl(comm := fbComm);
	AzimuthControl		: FB_AzimuthControl(comm := fbComm);
	TelescopeControl	: FB_MonetTelescopeControl(comm := fbComm);
	TelescopeAuxiliary  : FB_TelescopeAuxiliary(comm := fbComm);
	PendantControl		: FB_MonetPendantControl(comm := fbComm);
	
	//fbWeather			: FB_WeatherCheck();
	
	MqttWatchdog		: FB_MonetMqttWatchdog(comm := fbComm);	// park + close roof after 30 s without broker (MONETcommon)
	Diagnostics			: FB_MonetDiagnostics(comm := fbComm);	// diagnostics/base/* telemetry, on change + 30 s heartbeat (MONETcommon)
END_VAR
VAR CONSTANT
	telescopeConfig		: ST_TelescopeConfig := (longitude := 20.810808, latitude := -32.375823, altitude := 1798.0, 
												 azimuthPark := 175, elevationPark := 60, derotatorPark := 0, focusPark := 36.0, 
												 azimuthHome := 175, elevationHome := 40, derotatorHome := 0,
												 name := 'MONET/S', diameter := 1.2, cabinet := 'Beckhoff', manufacturer := 'Halfmann, Haidenhain, Beckhoff',
												 mountOptions := 'ALT-AZ', mount := 'ALT_AZ');
	fbPointing			: FB_PointingModelForward(AOFF := -0.006778523308102358, BNP := 0.030459575443670728, AN_A := -0.013961935190411667, AE_A := -0.01036163798027645, NPAE := 0.0017131069293910839, 
                                                  EOFF := 0.04040337399598415, AN_E := -0.011190631316106092, AE_E := -0.009741636951375865, TF := 0.06450337748465318);
	fbPointingInverse	: FB_PointingModelInversion(fbPointing := fbPointing);
END_VAR

(* 
Main control loop
* Execute sub modules
* power management
* control panel switches and status lamps

* start switch activates Hydraulics and Trafo
* 
*)

// get hostname for MQTT connection
GetHostName(bExecute := executeHostName, sHostName => HostName);
executeHostName := FALSE;

// run cabinet
CabinetControl();

// telescope mode
IF CabinetControl.KeyLocal THEN
	eTelescopeMode := SEL(HydraulicsControl.Enable, E_TelescopeMode.off, E_TelescopeMode.manual);	
ELSE
	eTelescopeMode := E_TelescopeMode.automatic; 
END_IF

// in local mode we can start or stop hydraulics and open the brake
brakeClearing := TRUE;
IF eTelescopeMode = E_TelescopeMode.manual OR eTelescopeMode = E_TelescopeMode.off THEN
	IF CabinetControl.IsStartPushed() THEN
		HydraulicsControl.Enable := TRUE;
	END_IF
	IF CabinetControl.IsStopPushed() THEN
		HydraulicsControl.Enable := FALSE;
	END_IF
	brakeClearing := CabinetControl.AreBreakesCleared();
	HydraulicsControl.bOpenBrake := brakeClearing;
END_IF

// clear errors: SafetyHandling.resetRequest (see call below) toggles Restart/ErrAck,
// here the cabinet/pendant reset button also resets covers, hydraulics and, in automatic mode, the
// telescope control (the only way to clear a latched bInterrupted)
IF CabinetControl.IsResetPushed() OR PendantControl.IbResetButton THEN
	CoverControl.Reset();
	HydraulicsControl.Reset();
	IF eTelescopeMode = E_TelescopeMode.automatic THEN
		TelescopeControl.Reset();
	END_IF
END_IF

// telescope is ready when power available
PowerMonitoring(phaseOK => ready);

// only run TelescopeControl in automatic mode
IF eTelescopeMode = E_TelescopeMode.automatic THEN
	TelescopeControl(
		telescopeConfig := telescopeConfig,
		fbCovers 		:= CoverControl,
		fbBrake 		:= HydraulicsControl,
		fbHydraulics 	:= HydraulicsControl,
		fbFocus 		:= FocusControl,
		fbElevation 	:= ElevationControl,
		fbAzimuth 		:= AzimuthControl,
		fbDerotator 	:= DerotatorControl,
		fbPointing      := fbPointing,
		fbPointingInverse := fbPointingInverse,
		bEstopTriggered := SafetyHandling.estop,	// M5: was never wired, see MONETcommon#11
		bMainReady		:= ready					// M5: was computed and published but never wired, see MONETcommon#11
	);
END_IF
TelescopeAuxiliary();

// run all control FBs
CoverControl();
HydraulicsControl(
	nMinPanLevel	:= 3500,
	nMaxPanLevel	:= 10200,
	fMinPanPercent	:= 0.0,
	fMaxPanPercent	:= 50.0, //56.0,
	bBrakeClearing	:= brakeClearing
);
ElevationControl(
	fCalibPosition 	:= 60.567917554230512,
	fbCovers 		:= CoverControl, 
	fbBrake 		:= HydraulicsControl
);
AzimuthControl(
	fCalibPosition	:= 1.1466144421902693,
	fMinPosition	:= -274.0,
	fMaxPosition	:= 270.0,
	bBrakeOpen		:= HydraulicsControl.brakeOpen,
);
DerotatorControl(
	fMinPosition		:= -90.0,
	fMaxPosition		:= 360.0
);	//
FocusControl(
	eTelescopeMode 	:= eTelescopeMode,
	fHomingPosition	:= 92.02, // 104.02 - 12.00
	fVelocity		:= 0.2,
	ptBrakeDelay	:= T#30S,
	ptFocusDelay	:= T#100MS
);
RoofControl(
	min_speed		:= 10000,
	max_speed 		:= 30000, 
	acceleration 	:= 150,
	max_position_1 	:= 205,
	max_position_2 	:= 203,
	max_position_diff	:= 3,
	limit_slowdown	:= 5
);
PendantControl(
	fbCovers 		:= CoverControl, 
	fbBrake 		:= HydraulicsControl, 
	fbHydraulics 	:= HydraulicsControl, 
	fbFocus 		:= FocusControl, 
	fbElevation 	:= ElevationControl, 
	fbAzimuth 		:= AzimuthControl, 
	fbDerotator 	:= DerotatorControl	
);

// MQTT watchdog: if connection is lost for more than the timeout, park and close roof.
// Armed only after the first successful connect -- otherwise a normal boot (bConnected
// starts FALSE until the initial hostname/connect/subscribe sequence completes) would
// trip this on every restart, not just real outages.
MqttWatchdog(bConnected := fbComm.bConnected, iTelescope := TelescopeControl, iRoof := RoofControl);

// and fbComm
fbComm(	
	sHostName		:= '192.168.127.10',
    nHostPort  		:= 1883,
    nKeepAlive  	:= 60,
	sTopicSub  		:= 'MONETS/Telescope/SET',
	sTopicPublish	:= 'MONETS/Telemetry',
	sTopicLog		:= 'MONETS/Log',
	Telescope		:= TelescopeControl,
	AltAzTelescope  := TelescopeControl,
	Focus			:= FocusControl,
	Roof			:= RoofControl
);

// check weather and UPSs
//fbWeather(
//	sHostName		:= '192.168.127.10',
//	nHostPort       := 8002,
//	sUri			:= '/api/current/'
//);
//IF fbWeather.bError OR NOT fbWeather.bWeatherGood THEN
	//TelescopeControl.Park();
	//RoofControl.Close();
//END_IF

// set control lights
//error := Focuscontrol.Error OR CoverControl.Error OR HydraulicsControl.Error;
error := CoverControl.Error OR HydraulicsControl.Error;
CabinetControl.SetManualLamp(eTelescopeMode = E_TelescopeMode.manual);

// blink errors
IF SafetyHandling.error THEN
	CabinetControl.SetBlinkError(E_Blink.short);
ELSIF ElevationControl.bError OR AzimuthControl.bError OR DerotatorControl.bError THEN
	CabinetControl.SetBlinkError(E_Blink.long);
ELSIF HydraulicsControl.bOilWarning OR HydraulicsControl.bOilHot OR HydraulicsControl.bPressureFailure THEN
	CabinetControl.SetBlinkError(E_Blink.slow);
ELSIF error THEN
	CabinetControl.SetBlinkError(E_Blink.on);
ELSE
	CabinetControl.SetBlinkError(E_Blink.off); 
END_IF

// power lamp is always on
CabinetControl.SetBlinkPower(E_Blink.on);

// do safety
SafetyHandling(resetRequest := CabinetControl.IsResetPushed() OR PendantControl.IbResetButton);

// telemetry
commTimer(IN:=TRUE);
IF commTimer.Q THEN
	commTimer(IN:=FALSE);
	fbComm.Publish('electronics', 'base', 'MainReady', BOOL_TO_STRING(ready));
	fbComm.Publish('electronics', 'base', 'MasterError', BOOL_TO_STRING(error));
	TelescopeAuxiliary.SendTelemetry();
END_IF

// diagnostics telemetry: publish on change, plus a full-snapshot heartbeat (MONETcommon)
Diagnostics(
	fbTelescope	:= TelescopeControl,
	fbElevation	:= ElevationControl,
	fbAzimuth	:= AzimuthControl,
	fbDerotator	:= DerotatorControl,
	fbFocus		:= FocusControl,
	fbSafety	:= SafetyHandling
);

END_PROGRAM

// ---- GlobalTextList.TcGTLO
TEXTLIST GlobalTextList
  4 = '%.0f'
  265 = '%.0f %'
  500 = '%.0f%'
  194 = '%.2f'
  730 = '%.2f mm'
  1120 = '%.2f °'
  943 = '%.2f °/s'
  1152 = '%.2f°'
  465 = '%.2f°/s'
  234 = '%.4'
  1272 = '%.4 °'
  484 = '%.4f'
  144 = '%.4f '
  339 = '%.4f mm'
  848 = '%.4f °'
  941 = '%.4f°'
  616 = '%d'
  792 = '%s'
  78 = '+'
  114 = '-'
  170 = '/'
  643 = '22'
  411 = 'Alt'
  207 = 'Altitude'
  148 = 'Automatic'
  1021 = 'Azimuth'
  785 = 'Azimuth:'
  247 = 'Brake'
  911 = 'Brake clearing'
  798 = 'Brake closed'
  396 = 'Brake open'
  958 = 'Brakes'
  272 = 'busy'
  573 = 'Busy'
  619 = 'Calculated'
  688 = 'Calibrated'
  337 = 'Close'
  41 = 'Close brake'
  507 = 'Closed'
  361 = 'Closing'
  392 = 'Cold'
  12 = 'Cover 1'
  678 = 'Cover 2'
  857 = 'Cover 3'
  816 = 'Current'
  1081 = 'Declination'
  815 = 'Derotator:'
  524 = 'Diag: %s'
  957 = 'Direction error'
  511 = 'Drive   Error'
  101 = 'EL1904'
  761 = 'EL2904'
  409 = 'Elevation:'
  894 = 'Enable'
  686 = 'EnabParkle'
  562 = 'Equatorial'
  868 = 'ErrAck'
  879 = 'Error'
  225 = 'Estop: %s'
  755 = 'Far'
  479 = 'Global'
  548 = 'GoHome'
  867 = 'GoTo'
  331 = 'High'
  940 = 'Homed'
  483 = 'Homing'
  1063 = 'Horizontal'
  81 = 'Hot'
  163 = 'Level'
  846 = 'Level:'
  728 = 'Limit error'
  363 = 'Limiterror'
  557 = 'Limits'
  58 = 'Low'
  697 = 'Manual'
  389 = 'Motor #1'
  611 = 'Motor #2'
  712 = 'Move'
  466 = 'Movement'
  765 = 'Moving'
  59 = 'Near'
  33 = 'Oil cold'
  995 = 'Oil high'
  856 = 'Oil hot'
  768 = 'Oil low'
  37 = 'Oil pan maximum'
  481 = 'Oil pressure OK'
  874 = 'Oil Status'
  498 = 'Oil warning'
  366 = 'Open'
  482 = 'Open brake'
  1197 = 'Open/Close'
  186 = 'Opening'
  352 = 'Override Start Pump'
  744 = 'Override Start Sucction'
  606 = 'Override stop pump'
  890 = 'Overrides'
  384 = 'Pan max'
  273 = 'park'
  92 = 'Park'
  1353 = 'Parked'
  525 = 'Position'
  919 = 'Power'
  641 = 'Pressure'
  196 = 'Pump'
  523 = 'Pump running'
  120 = 'ready'
  176 = 'Ready'
  685 = 'Reset'
  789 = 'Restart'
  1221 = 'Right Ascension'
  360 = 'Roof'
  456 = 'Roof #1'
  944 = 'Roof #2'
  104 = 'Safety Diag%s'
  521 = 'Safety Diag: %s'
  672 = 'Safety State: %s'
  309 = 'Set'
  777 = 'slew'
  1245 = 'Slew'
  724 = 'Slewing'
  717 = 'sliding'
  138 = 'Slow close'
  996 = 'Slow open'
  49 = 'Speed'
  566 = 'Start'
  202 = 'Start Sucction'
  27 = 'Start suction'
  520 = 'State'
  809 = 'State: %s'
  354 = 'Status'
  328 = 'STO ErrAck:'
  540 = 'STO Reset:'
  488 = 'STO:'
  572 = 'Stop'
  189 = 'Stop pump'
  155 = 'stopped'
  790 = 'Stopped'
  614 = 'Sucction'
  782 = 'Sucction running'
  704 = 'Succtionrunning'
  552 = 'Suction'
  385 = 'Sync error'
  362 = 'track'
  569 = 'Track'
  364 = 'tracking'
  356 = 'Tracking'
  136 = 'Unlocked'
  67 = 'Velocity'
  480 = 'Warning'
  609 = 'Zero counter'
  1015 = ']'
END_TEXTLIST

// ---- VISUs/Azimuth.TcVIS
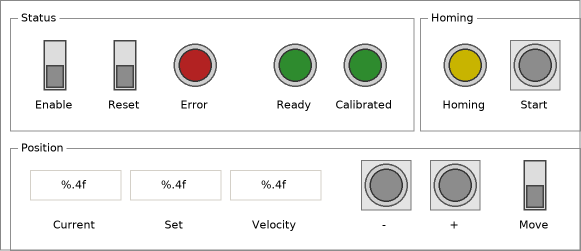
VISUALIZATION Azimuth  // 581x251
    GroupBox (10,10 404x121), "Status"
        DipSwitch (20,30 50x50), variable: MAIN.AzimuthControl.bEnable, behaviour: TOGGLE, style: Switch-DipSwitch-Gray
        DipSwitch (90,30 50x50), variable: MAIN.AzimuthControl.bReset, behaviour: TOGGLE, style: Switch-DipSwitch-Gray
        Lamp1 (160,30 50x50), variable: MAIN.AzimuthControl.bError, style: Lamp-Lamp1-Red
        Lamp1 (260,30 50x50), variable: MAIN.AzimuthControl.bReady, style: Lamp-Lamp1-Green
        Lamp1 (330,30 50x50), variable: MAIN.AzimuthControl.bCalibrated, style: Lamp-Lamp1-Green
        Label (10,80 68x30), "Enable"
        Label (80,80 68x30), "Reset"
        Label (150,80 68x30), "Error"
        Label (250,80 68x30), "Ready"
        Label (320,80 68x30), "Calibrated"
    GroupBox (420,10 161x121), "Homing"
        Lamp1 (20,30 50x50), variable: MAIN.AzimuthControl.bHomeAxis, style: Lamp-Lamp1-Yellow
        Label (10,80 68x30), "Homing"
        PushSwitch (90,30 50x50), variable: MAIN.AzimuthControl.bHomeAxis, behaviour: TOGGLE, style: Switch-PushSwitch-Gray
        Label (80,80 68x30), "Start"
    GroupBox (10,140 571x111), "Position"
        Textfield (20,30 91x30), "%.4f", text variable: MAIN.AzimuthControl.fActualPosition
        Label (30,70 68x30), "Current"
        Textfield (120,30 91x30), "%.4f", text variable: MAIN.AzimuthControl.fPosition
            OnMouseUp: write the text variable via InputWithLimits, min MAIN.AzimuthControl.fMinPosition, max MAIN.AzimuthControl.fMaxPosition
        Textfield (220,30 91x30), "%.4f", text variable: MAIN.AzimuthControl.fVelocity
            OnMouseUp: write the text variable via InputWithLimits, min 0, max 200
        PushSwitch (351,20 50x50), variable: MAIN.AzimuthControl.bMoveNeg, behaviour: TOGGLE, style: Switch-PushSwitch-Gray
        PushSwitch (420,20 50x50), variable: MAIN.AzimuthControl.bMovePos, behaviour: TOGGLE, style: Switch-PushSwitch-Gray
        DipSwitch (500,20 50x50), variable: MAIN.AzimuthControl.bMoveAxis, behaviour: TOGGLE, style: Switch-DipSwitch-Gray
        Label (340,70 68x30), "-"
        Label (410,70 68x30), "+"
        Label (490,70 68x30), "Move"
    Label (140,210 68x30), "Set"
    Label (240,210 68x30), "Velocity"
END_VISUALIZATION

// ---- VISUs/Cover.TcVIS
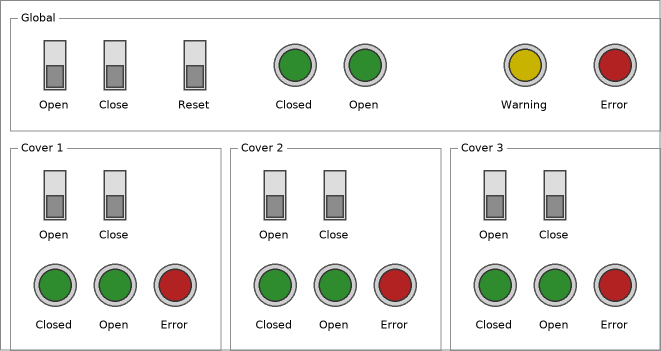
VISUALIZATION Cover  // 661x351
    GroupBox (10,10 651x121), "Global"
        DipSwitch (20,30 50x50), variable: MAIN.CoverControl.bOpen, behaviour: TOGGLE, style: Switch-DipSwitch-Gray
        DipSwitch (80,30 50x50), variable: MAIN.CoverControl.bClose, behaviour: TOGGLE, style: Switch-DipSwitch-Gray
        Lamp1 (260,30 50x50), variable: MAIN.CoverControl.bAllClosed, style: Lamp-Lamp1-Green
        Lamp1 (330,30 50x50), variable: MAIN.CoverControl.bAllOpen, style: Lamp-Lamp1-Green
        Label (10,80 68x30), "Open"
        Label (70,80 68x30), "Close"
        Label (250,80 68x30), "Closed"
        Label (320,80 68x30), "Open"
        DipSwitch (160,30 50x50), variable: MAIN.CoverControl.bReset, behaviour: TOGGLE, style: Switch-DipSwitch-Gray
        Lamp1 (490,30 50x50), variable: MAIN.CoverControl.bWarning, style: Lamp-Lamp1-Yellow
        Lamp1 (580,30 50x50), variable: MAIN.CoverControl.bError, style: Lamp-Lamp1-Red
        Label (570,80 68x30), "Error"
        Label (480,80 68x30), "Warning"
    GroupBox (10,140 211x211), "Cover 1"
        Label (130,170 68x30), "Error"
        Lamp1 (20,120 50x50), variable: MAIN.CoverControl.abCoverClosed[1], style: Lamp-Lamp1-Green
        Lamp1 (80,120 50x50), variable: MAIN.CoverControl.abCoverOpen[1], style: Lamp-Lamp1-Green
        Label (10,170 68x30), "Closed"
        Label (70,170 68x30), "Open"
        DipSwitch (20,30 50x50), variable: MAIN.CoverControl.OabOpenCover[1], behaviour: TOGGLE, style: Switch-DipSwitch-Gray
        DipSwitch (80,30 50x50), variable: MAIN.CoverControl.OabCloseCover[1], behaviour: TOGGLE, style: Switch-DipSwitch-Gray
        Label (10,80 68x30), "Open"
        Label (70,80 68x30), "Close"
        Lamp1 (140,120 50x50), variable: MAIN.CoverControl.abCoverError[1], style: Lamp-Lamp1-Red
    Label (160,90 68x30), "Reset"
    GroupBox (230,140 211x211), "Cover 2"
        Label (130,170 68x30), "Error"
        Lamp1 (20,120 50x50), variable: MAIN.CoverControl.abCoverClosed[2], style: Lamp-Lamp1-Green
        Lamp1 (80,120 50x50), variable: MAIN.CoverControl.abCoverOpen[2], style: Lamp-Lamp1-Green
        Label (10,170 68x30), "Closed"
        Label (70,170 68x30), "Open"
        DipSwitch (20,30 50x50), variable: MAIN.CoverControl.OabOpenCover[2], behaviour: TOGGLE, style: Switch-DipSwitch-Gray
        DipSwitch (80,30 50x50), variable: MAIN.CoverControl.OabCloseCover[2], behaviour: TOGGLE, style: Switch-DipSwitch-Gray
        Label (10,80 68x30), "Open"
        Label (70,80 68x30), "Close"
        Lamp1 (140,120 50x50), variable: MAIN.CoverControl.abCoverError[2], style: Lamp-Lamp1-Red
    GroupBox (450,140 211x211), "Cover 3"
        Label (130,170 68x30), "Error"
        Lamp1 (20,120 50x50), variable: MAIN.CoverControl.abCoverClosed[3], style: Lamp-Lamp1-Green
        Lamp1 (80,120 50x50), variable: MAIN.CoverControl.abCoverOpen[3], style: Lamp-Lamp1-Green
        Label (10,170 68x30), "Closed"
        Label (70,170 68x30), "Open"
        DipSwitch (20,30 50x50), variable: MAIN.CoverControl.OabOpenCover[3], behaviour: TOGGLE, style: Switch-DipSwitch-Gray
        DipSwitch (80,30 50x50), variable: MAIN.CoverControl.OabCloseCover[3], behaviour: TOGGLE, style: Switch-DipSwitch-Gray
        Label (10,80 68x30), "Open"
        Label (70,80 68x30), "Close"
        Lamp1 (140,120 50x50), variable: MAIN.CoverControl.abCoverError[3], style: Lamp-Lamp1-Red
END_VISUALIZATION

// ---- VISUs/Derotator.TcVIS
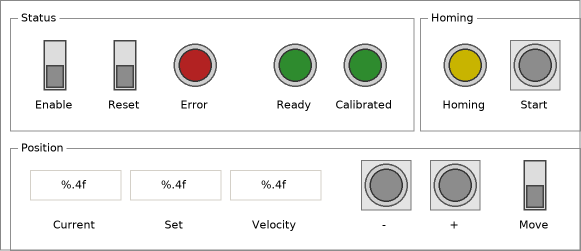
VISUALIZATION Derotator  // 581x251
    GroupBox (10,10 404x121), "Status"
        DipSwitch (20,30 50x50), variable: MAIN.DerotatorControl.bEnable, behaviour: TOGGLE, style: Switch-DipSwitch-Gray
        DipSwitch (90,30 50x50), variable: MAIN.DerotatorControl.bReset, behaviour: TOGGLE, style: Switch-DipSwitch-Gray
        Lamp1 (160,30 50x50), variable: MAIN.DerotatorControl.bError, style: Lamp-Lamp1-Red
        Lamp1 (260,30 50x50), variable: MAIN.DerotatorControl.bReady, style: Lamp-Lamp1-Green
        Lamp1 (330,30 50x50), variable: MAIN.DerotatorControl.bCalibrated, style: Lamp-Lamp1-Green
        Label (10,80 68x30), "Enable"
        Label (80,80 68x30), "Reset"
        Label (150,80 68x30), "Error"
        Label (250,80 68x30), "Ready"
        Label (320,80 68x30), "Calibrated"
    GroupBox (420,10 161x121), "Homing"
        Lamp1 (20,30 50x50), variable: MAIN.DerotatorControl.bHomeAxis, style: Lamp-Lamp1-Yellow
        Label (10,80 68x30), "Homing"
        PushSwitch (90,30 50x50), variable: MAIN.DerotatorControl.bHomeAxis, behaviour: TOGGLE, style: Switch-PushSwitch-Gray
        Label (80,80 68x30), "Start"
    GroupBox (10,140 571x111), "Position"
        Textfield (20,30 91x30), "%.4f", text variable: MAIN.DerotatorControl.fActualPosition
        Label (30,70 68x30), "Current"
        Textfield (120,30 91x30), "%.4f", text variable: MAIN.DerotatorControl.fPosition
            OnMouseUp: write the text variable via InputWithLimits, min MAIN.DerotatorControl.fMinPosition, max MAIN.DerotatorControl.fMaxPosition
        Textfield (220,30 91x30), "%.4f", text variable: MAIN.DerotatorControl.fVelocity
            OnMouseUp: write the text variable via InputWithLimits, min 0, max 200
        PushSwitch (351,20 50x50), variable: MAIN.DerotatorControl.bMoveNeg, behaviour: TOGGLE, style: Switch-PushSwitch-Gray
        PushSwitch (420,20 50x50), variable: MAIN.DerotatorControl.bMovePos, behaviour: TOGGLE, style: Switch-PushSwitch-Gray
        DipSwitch (500,20 50x50), variable: MAIN.DerotatorControl.bMoveAxis, behaviour: TOGGLE, style: Switch-DipSwitch-Gray
        Label (340,70 68x30), "-"
        Label (410,70 68x30), "+"
        Label (490,70 68x30), "Move"
    Label (140,210 68x30), "Set"
    Label (240,210 68x30), "Velocity"
END_VISUALIZATION

// ---- VISUs/Elevation.TcVIS
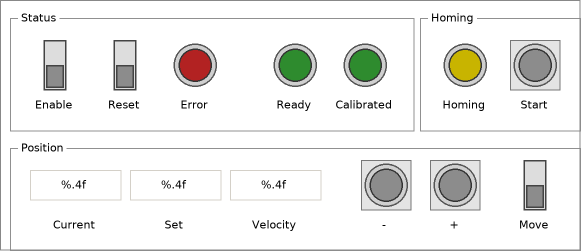
VISUALIZATION Elevation  // 581x251
    GroupBox (10,10 404x121), "Status"
        DipSwitch (20,30 50x50), variable: MAIN.ElevationControl.bEnable, behaviour: TOGGLE, style: Switch-DipSwitch-Gray
        DipSwitch (90,30 50x50), variable: MAIN.ElevationControl.bReset, behaviour: TOGGLE, style: Switch-DipSwitch-Gray
        Lamp1 (160,30 50x50), variable: MAIN.ElevationControl.bError, style: Lamp-Lamp1-Red
        Lamp1 (260,30 50x50), variable: MAIN.ElevationControl.bReady, style: Lamp-Lamp1-Green
        Lamp1 (330,30 50x50), variable: MAIN.ElevationControl.bCalibrated, style: Lamp-Lamp1-Green
        Label (10,80 68x30), "Enable"
        Label (80,80 68x30), "Reset"
        Label (150,80 68x30), "Error"
        Label (250,80 68x30), "Ready"
        Label (320,80 68x30), "Calibrated"
    GroupBox (420,10 161x121), "Homing"
        Lamp1 (20,30 50x50), variable: MAIN.ElevationControl.bHomeAxis, style: Lamp-Lamp1-Yellow
        Label (10,80 68x30), "Homing"
        PushSwitch (90,30 50x50), variable: MAIN.ElevationControl.bHomeAxis, behaviour: TOGGLE, style: Switch-PushSwitch-Gray
        Label (80,80 68x30), "Start"
    GroupBox (10,140 571x111), "Position"
        Textfield (20,30 91x30), "%.4f", text variable: MAIN.ElevationControl.fActualPosition
        Label (30,70 68x30), "Current"
        Textfield (120,30 91x30), "%.4f", text variable: MAIN.ElevationControl.fPosition
            OnMouseUp: write the text variable via InputWithLimits, min MAIN.ElevationControl.fMinPosition, max MAIN.ElevationControl.fMaxPosition
        Textfield (220,30 91x30), "%.4f", text variable: MAIN.ElevationControl.fVelocity
            OnMouseUp: write the text variable via InputWithLimits, min 0, max 200
        PushSwitch (351,20 50x50), variable: MAIN.ElevationControl.bMoveNeg, behaviour: TOGGLE, style: Switch-PushSwitch-Gray
        PushSwitch (420,20 50x50), variable: MAIN.ElevationControl.bMovePos, behaviour: TOGGLE, style: Switch-PushSwitch-Gray
        DipSwitch (500,20 50x50), variable: MAIN.ElevationControl.bMoveAxis, behaviour: TOGGLE, style: Switch-DipSwitch-Gray
        Label (340,70 68x30), "-"
        Label (410,70 68x30), "+"
        Label (490,70 68x30), "Move"
    Label (140,210 68x30), "Set"
    Label (240,210 68x30), "Velocity"
END_VISUALIZATION

// ---- VISUs/Focus.TcVIS
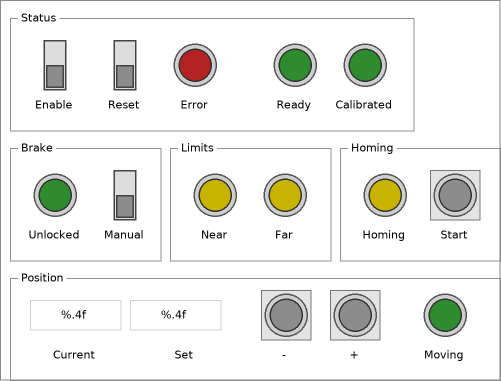
VISUALIZATION Focus  // 501x381
    GroupBox (10,10 404x121), "Status"
        DipSwitch (20,30 50x50), variable: MAIN.FocusControl.bEnable, behaviour: TOGGLE, style: Switch-DipSwitch-Gray
        DipSwitch (90,30 50x50), variable: MAIN.FocusControl.bReset, behaviour: TOGGLE, style: Switch-DipSwitch-Gray
        Lamp1 (160,30 50x50), variable: MAIN.FocusControl.bError, style: Lamp-Lamp1-Red
        Lamp1 (260,30 50x50), variable: MAIN.FocusControl.bReady, style: Lamp-Lamp1-Green
        Lamp1 (330,30 50x50), variable: MAIN.FocusControl.bCalibrated, style: Lamp-Lamp1-Green
        Label (10,80 68x30), "Enable"
        Label (80,80 68x30), "Reset"
        Label (150,80 68x30), "Error"
        Label (250,80 68x30), "Ready"
        Label (320,80 68x30), "Calibrated"
        Lamp1 (410,280 50x50), variable: MAIN.AzimuthControl.bCalibrated, style: Lamp-Lamp1-Green
    GroupBox (340,140 161x121), "Homing"
        Lamp1 (20,30 50x50), variable: MAIN.FocusControl.bHomeAxis, style: Lamp-Lamp1-Yellow
        Label (10,80 68x30), "Homing"
        PushSwitch (90,30 50x50), variable: MAIN.FocusControl.bHomeAxis, behaviour: TOGGLE, style: Switch-PushSwitch-Gray
        Label (80,80 68x30), "Start"
    GroupBox (10,140 151x121), "Brake"
        DipSwitch (90,30 50x50), variable: MAIN.FocusControl.bManualUnlock, behaviour: TOGGLE, style: Switch-DipSwitch-Gray
        Lamp1 (20,30 50x50), variable: MAIN.FocusControl.bFocusUnlocked, style: Lamp-Lamp1-Green
        Label (80,80 68x30), "Manual"
        Label (10,80 68x30), "Unlocked"
    GroupBox (170,140 161x121), "Limits"
        Lamp1 (20,30 50x50), variable: MAIN.FocusControl.IbLimitNear, style: Lamp-Lamp1-Yellow
        Label (10,80 68x30), "Near"
        Lamp1 (90,30 50x50), variable: MAIN.FocusControl.IbLimitFar, style: Lamp-Lamp1-Yellow
    Label (250,220 68x30), "Far"
    GroupBox (10,270 491x111), "Position"
        Textfield (20,30 91x30), "%.4f", text variable: MAIN.FocusControl.fActualPosition
        Label (30,70 68x30), "Current"
        Textfield (120,30 91x30), "%.4f", text variable: MAIN.FocusControl.fPosition
            OnMouseUp: write the text variable via InputWithLimits, min MAIN.AzimuthControl.fMinPosition, max MAIN.AzimuthControl.fMaxPosition
        PushSwitch (251,20 50x50), variable: MAIN.FocusControl.bMoveNeg, behaviour: TOGGLE, style: Switch-PushSwitch-Gray
        PushSwitch (320,20 50x50), variable: MAIN.FocusControl.bMovePos, behaviour: TOGGLE, style: Switch-PushSwitch-Gray
        Label (240,70 68x30), "-"
        Label (310,70 68x30), "+"
        Label (140,70 68x30), "Set"
        Lamp1 (410,20 50x50), variable: MAIN.FocusControl.bMoveAxis, style: Lamp-Lamp1-Green
    Label (410,340 68x30), "Moving"
END_VISUALIZATION

// ---- VISUs/Hydraulics.TcVIS
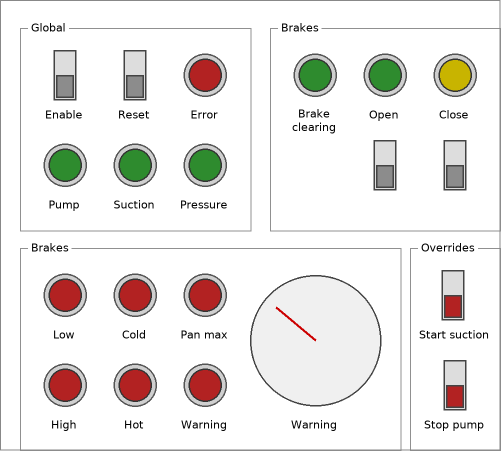
VISUALIZATION Hydraulics  // 501x451
    GroupBox (20,20 231x211), "Global"
        DipSwitch (20,30 50x50), variable: MAIN.HydraulicsControl.bEnable, behaviour: TOGGLE, style: Switch-DipSwitch-Gray
        DipSwitch (90,30 50x50), variable: MAIN.HydraulicsControl.bReset, behaviour: TOGGLE, style: Switch-DipSwitch-Gray
        Lamp1 (160,30 50x50), variable: MAIN.HydraulicsControl.bError, style: Lamp-Lamp1-Red
        Lamp1 (20,120 50x50), variable: MAIN.HydraulicsControl.bPumpRunning, style: Lamp-Lamp1-Green
        Lamp1 (90,120 50x50), variable: MAIN.HydraulicsControl.bSuctionRunning, style: Lamp-Lamp1-Green
        Label (10,80 68x30), "Enable"
        Label (80,80 68x30), "Reset"
        Label (150,80 68x30), "Error"
        Label (10,170 68x30), "Pump"
        Label (80,170 68x30), "Suction"
        Lamp1 (160,120 50x50), variable: MAIN.HydraulicsControl.bOilPressureOK, style: Lamp-Lamp1-Green
        Label (150,170 68x30), "Pressure"
    GroupBox (270,20 231x211), "Brakes"
        DipSwitch (90,120 50x50), variable: MAIN.HydraulicsControl.bOpenBrake, behaviour: TOGGLE, style: Switch-DipSwitch-Gray
        DipSwitch (160,120 50x50), variable: MAIN.HydraulicsControl.bCloseBrake, behaviour: TOGGLE, style: Switch-DipSwitch-Gray
        Lamp1 (160,30 50x50), variable: MAIN.HydraulicsControl.bBrakeClosed, style: Lamp-Lamp1-Yellow
        Lamp1 (20,30 50x50), variable: MAIN.HydraulicsControl.bBrakeClearing, style: Lamp-Lamp1-Green
        Label (150,80 68x30), "Close"
        Label (10,80 68x41), "Brake clearing"
        Lamp1 (90,30 50x50), variable: MAIN.HydraulicsControl.bBrakeOpen, style: Lamp-Lamp1-Green
        Label (80,80 68x30), "Open"
    GroupBox (20,240 381x211), "Brakes"
        Lamp1 (160,30 50x50), variable: MAIN.HydraulicsControl.bOilPanMaximum, style: Lamp-Lamp1-Red
        Label (150,80 68x30), "Pan max"
        Lamp1 (20,30 50x50), variable: MAIN.HydraulicsControl.bOilLow, style: Lamp-Lamp1-Red
        Lamp1 (90,30 50x50), variable: MAIN.HydraulicsControl.bOilCold, style: Lamp-Lamp1-Red
        Label (80,80 68x30), "Cold"
        Label (10,80 68x30), "Low"
        Lamp1 (160,120 50x50), variable: MAIN.HydraulicsControl.bOilWarning, style: Lamp-Lamp1-Red
        Meter360 (230,30 131x141), value: MAIN.HydraulicsControl.fOilLevel, style: Meter-Meter360-Gray, scale format: %.0f, scale 0..120
        Label (260,170 68x30), "Warning"
    Label (170,410 68x30), "Warning"
    Lamp1 (40,360 50x50), variable: MAIN.HydraulicsControl.bOilHigh, style: Lamp-Lamp1-Red
    Lamp1 (110,360 50x50), variable: MAIN.HydraulicsControl.bOilHot, style: Lamp-Lamp1-Red
    Label (100,410 68x30), "Hot"
    Label (30,410 68x30), "High"
    GroupBox (410,240 91x211), "Overrides"
        DipSwitch (18,30 50x50), variable: MAIN.HydraulicsControl.bManualSuction, behaviour: TOGGLE, style: Switch-DipSwitch-Red
        DipSwitch (20,120 50x50), variable: MAIN.HydraulicsControl.bManualPumpStop, behaviour: TOGGLE, style: Switch-DipSwitch-Red
        Label (10,80 68x30), "Start suction"
        Label (10,170 68x30), "Stop pump"
END_VISUALIZATION

// ---- VISUs/Pendant.TcVIS
VISUALIZATION Pendant  // 1024x768
END_VISUALIZATION

// ---- VISUs/Safety.TcVIS
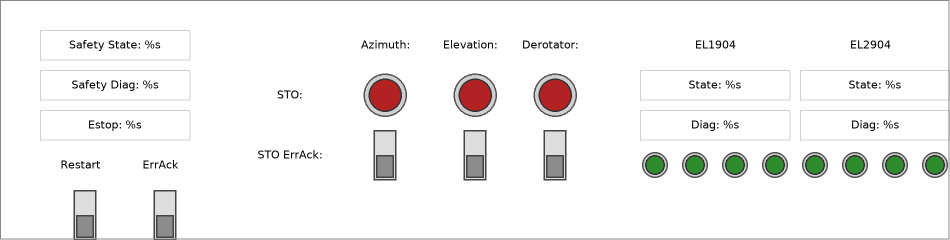
VISUALIZATION Safety  // 950x240
    Label (340,30 91x30), "Azimuth:"
    Lamp1 (360,70 50x50), variable: MAIN.AzimuthControl.IbSTO, style: Lamp-Lamp1-Red
    Label (430,30 81x30), "Elevation:"
    Lamp1 (450,70 50x50), variable: MAIN.ElevationControl.IbSTO, style: Lamp-Lamp1-Red
    Label (510,30 81x30), "Derotator:"
    Lamp1 (530,70 50x50), variable: MAIN.DerotatorControl.IbSTO, style: Lamp-Lamp1-Red
    Label (240,80 100x30), "STO:"
    DipSwitch (60,190 50x50), variable: MAIN.SafetyHandling.outRestart, behaviour: TOGGLE, style: Switch-DipSwitch-Gray
    DipSwitch (530,130 50x50), variable: MAIN.SafetyHandling.outResetDerotatorSTO, behaviour: TOGGLE, style: Switch-DipSwitch-Gray
    DipSwitch (360,130 50x50), variable: MAIN.SafetyHandling.outResetAzimuthSTO, behaviour: TOGGLE, style: Switch-DipSwitch-Gray
    DipSwitch (450,130 50x50), variable: MAIN.SafetyHandling.outResetElevationSTO, behaviour: TOGGLE, style: Switch-DipSwitch-Gray
    Label (240,140 100x30), "STO ErrAck:"
    Label (40,150 81x30), "Restart"
    DipSwitch (140,190 50x50), variable: MAIN.SafetyHandling.outErrAck, behaviour: TOGGLE, style: Switch-DipSwitch-Gray
    Label (120,150 81x30), "ErrAck"
    Textfield (40,30 150x30), "Safety State: %s", text variable: MAIN.SafetyHandling.fbInfoEStop1.sState, input disabled if: TRUE
    Textfield (40,110 150x30), "Estop: %s", text variable: MAIN.SafetyHandling.fbInfoEStop1.sState, input disabled if: TRUE
    Textfield (40,70 150x30), "Safety Diag: %s", text variable: MAIN.SafetyHandling.fbInfoEStop1.sDiag, input disabled if: TRUE
    Label (670,30 91x30), "EL1904"
    Label (830,30 81x30), "EL2904"
    Textfield (640,70 150x30), "State: %s", text variable: MAIN.SafetyHandling.fbInfoSafetyIn.sState, input disabled if: TRUE
    Textfield (640,110 150x30), "Diag: %s", text variable: MAIN.SafetyHandling.fbInfoSafetyIn.sDiag, input disabled if: TRUE
    Textfield (800,70 150x30), "State: %s", text variable: MAIN.SafetyHandling.fbInfoSafetyOut.sState, input disabled if: TRUE
    Textfield (800,110 150x30), "Diag: %s", text variable: MAIN.SafetyHandling.fbInfoSafetyOut.sDiag, input disabled if: TRUE
    Lamp1 (640,150 30x30), variable: MAIN.SafetyHandling.bSafetyInCh1, style: Lamp-Lamp1-Green
    Lamp1 (680,150 30x30), variable: MAIN.SafetyHandling.bSafetyInCh2, style: Lamp-Lamp1-Green
    Lamp1 (720,150 30x30), variable: MAIN.SafetyHandling.bSafetyInCh3, style: Lamp-Lamp1-Green
    Lamp1 (760,150 30x30), variable: MAIN.SafetyHandling.bSafetyInCh4, style: Lamp-Lamp1-Green
    Lamp1 (800,150 30x30), variable: MAIN.SafetyHandling.bSafetyInCh1, style: Lamp-Lamp1-Green
    Lamp1 (840,150 30x30), variable: MAIN.SafetyHandling.bSafetyInCh2, style: Lamp-Lamp1-Green
    Lamp1 (880,150 30x30), variable: MAIN.SafetyHandling.bSafetyInCh3, style: Lamp-Lamp1-Green
    Lamp1 (920,150 30x30), variable: MAIN.SafetyHandling.bSafetyInCh4, style: Lamp-Lamp1-Green
END_VISUALIZATION

// ---- VISUs/Telescope.TcVIS
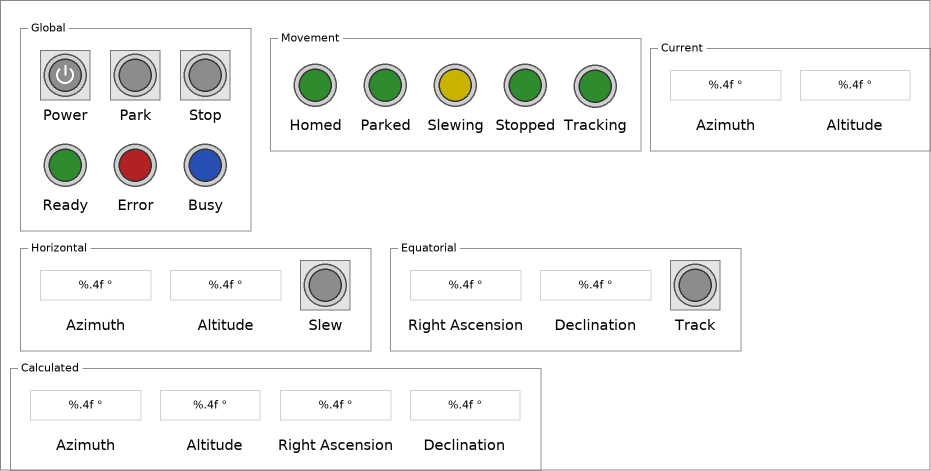
VISUALIZATION Telescope  // 931x471
    GroupBox (20,20 231x211), "Global"
        Label (0,80 91x30), "Power"
        Lamp1 (90,120 50x50), variable: MAIN.TelescopeControl.bError, style: Lamp-Lamp1-Red
        Label (90,170 51x30), "Error"
        Lamp1 (20,120 50x50), variable: MAIN.TelescopeControl.bReady, style: Lamp-Lamp1-Green
        Label (20,170 51x30), "Ready"
        PowerSwitch (20,30 50x50), variable: MAIN.TelescopeControl.bPower, behaviour: TOGGLE, style: Switch-PowerSwitch-Gray
        PushSwitch (90,30 50x50), variable: MAIN.TelescopeControl.bPark, behaviour: TOGGLE, style: Switch-PushSwitch-Gray
        Lamp1 (160,120 50x50), variable: MAIN.TelescopeControl.bBusy, style: Lamp-Lamp1-Blue
        Label (160,170 51x30), "Busy"
        PushSwitch (160,30 50x50), variable: MAIN.TelescopeControl.bPark, behaviour: TOGGLE, style: Switch-PushSwitch-Gray
        Label (140,80 91x30), "Stop"
    Label (90,100 91x30), "Park"
    GroupBox (20,240 351x111), "Horizontal"
        Label (30,70 91x30), "Azimuth"
        Textfield (20,30 111x30), "%.4f °", text variable: MAIN.TelescopeControl.fAzimuth
            OnMouseClick: write the text variable via InputWithLimits, min 0, max 360
        Label (160,70 91x30), "Altitude"
        PushSwitch (280,20 50x50), variable: MAIN.TelescopeControl.bSlew, behaviour: TOGGLE, style: Switch-PushSwitch-Gray
        Label (260,70 91x30), "Slew"
    Textfield (170,270 111x30), "%.4f °", text variable: MAIN.TelescopeControl.fElevation
        OnMouseClick: write the text variable via Default, min 0, max 90
    GroupBox (10,360 531x111), "Calculated"
        Label (30,70 91x30), "Azimuth"
        Textfield (20,30 111x30), "%.4f °", text variable: MAIN.TelescopeControl.fAzimuthCalc
        Label (159,70 91x30), "Altitude"
        Textfield (150,30 100x30), "%.4f °", text variable: MAIN.TelescopeControl.fElevationCalc
        Label (270,70 111x30), "Right Ascension"
        Textfield (270,30 111x30), "%.4f °", text variable: MAIN.TelescopeControl.fRightAscensionCalc
        Label (409,70 91x30), "Declination"
        Textfield (400,30 110x30), "%.4f °", text variable: MAIN.TelescopeControl.fDeclinationCalc
    GroupBox (650,40 281x111), "Current"
        Label (30,70 91x30), "Azimuth"
        Textfield (20,30 111x30), "%.4f °", text variable: MAIN.TelescopeControl.fAzimuthCurrent
        Label (159,70 91x30), "Altitude"
        Textfield (150,30 110x30), "%.4f °", text variable: MAIN.TelescopeControl.fElevationCurrent
    GroupBox (270,30 371x121), "Movement"
        Lamp1 (90,30 50x50), variable: MAIN.TelescopeControl.bIsParked, style: Lamp-Lamp1-Green
        Label (90,80 51x30), "Parked"
        Lamp1 (160,30 50x50), variable: MAIN.TelescopeControl.bSlewing, style: Lamp-Lamp1-Yellow
        Label (150,80 71x30), "Slewing"
        Lamp1 (230,30 50x50), variable: MAIN.TelescopeControl.bStopped, style: Lamp-Lamp1-Green
        Label (220,80 71x30), "Stopped"
        Lamp1 (300,31 50x50), variable: MAIN.TelescopeControl.bTracking, style: Lamp-Lamp1-Green
        Label (290,80 71x30), "Tracking"
        Lamp1 (20,30 50x50), variable: MAIN.TelescopeControl.bHomed, style: Lamp-Lamp1-Green
        Label (20,80 51x30), "Homed"
    GroupBox (390,240 351x111), "Equatorial"
        Label (20,70 111x30), "Right Ascension"
        Textfield (20,30 111x30), "%.4f °", text variable: MAIN.TelescopeControl.fRightAscension
            OnMouseClick: write the text variable via InputWithLimits, min 0, max 360
        Label (160,70 91x30), "Declination"
        PushSwitch (280,20 50x50), variable: MAIN.TelescopeControl.bGoto, behaviour: TOGGLE, style: Switch-PushSwitch-Gray
        Label (260,70 91x30), "Track"
        Textfield (150,30 111x30), "%.4f °", text variable: MAIN.TelescopeControl.fDeclination
            OnMouseClick: write the text variable via Default, min -90, max 90
END_VISUALIZATION

// ---- VISUs/Visualization.TcVIS
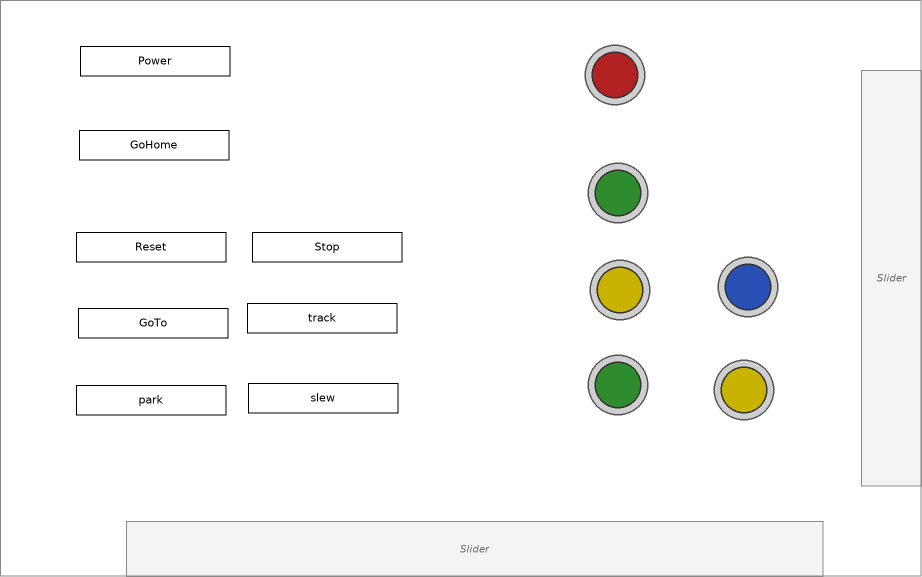
VISUALIZATION Visualization  // 922x577
    RoundedRectangle (80,46 150x30), "Power", colour toggle: TelescopeControl.power
        toggle TelescopeControl.power
    Rectangle (79,130 150x30), "GoHome", colour toggle: TelescopeControl.gohome
        toggle TelescopeControl.gohome
    Lamp1 (580,40 70x70), tooltip "Error", variable: TelescopeControl.error, style: Lamp-Lamp1-Red
    Lamp1 (583,158 70x70), tooltip "ready", variable: TelescopeControl.ready, style: Lamp-Lamp1-Green
    Rectangle (76,232 150x30), "Reset", colour toggle: TelescopeControl.reset
        toggle TelescopeControl.reset
    RoundedRectangle (78,308 150x30), "GoTo", colour toggle: TelescopeControl.goto
        toggle TelescopeControl.goto
    Lamp1 (585,255 70x70), tooltip "sliding", variable: TelescopeControl.sliding, style: Lamp-Lamp1-Yellow
    RoundedRectangle (76,385 150x30), "park", colour toggle: TelescopeControl.park
        toggle TelescopeControl.park
    Lamp1 (583,350 70x70), tooltip "stopped", variable: TelescopeControl.Safetypped, style: Lamp-Lamp1-Green
    Slider (126,521 697x56), variable: TelescopeControl.rightascension, scale 0..360
    Slider (861,70 61x416), variable: TelescopeControl.declination, scale -90..90
    Lamp1 (713,252 70x70), tooltip "tracking", variable: TelescopeControl.tracking, style: Lamp-Lamp1-Blue
    RoundedRectangle (247,303 150x30), "track", colour toggle: TelescopeControl.track
        toggle TelescopeControl.track
    RoundedRectangle (248,383 150x30), "slew", colour toggle: TelescopeControl.slew
        toggle TelescopeControl.slew
    Lamp1 (709,355 70x70), tooltip "busy", variable: TelescopeControl.busy, style: Lamp-Lamp1-Yellow
    RoundedRectangle (252,232 150x30), "Stop", colour toggle: TelescopeControl.Safetyp
        toggle TelescopeControl.stop
END_VISUALIZATION

// ---- VISUs/Roof.TcVIS
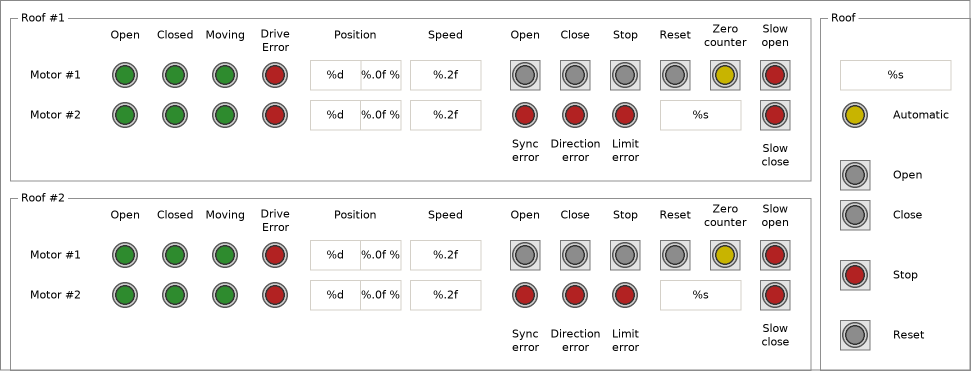
VISUALIZATION Roof  // 971x371
    GroupBox (10,10 801x171), "Roof #1"
        Label (10,50 71x30), "Motor #1"
        Label (10,90 71x30), "Motor #2"
        Label (80,10 71x30), "Open"
        Label (130,10 71x30), "Closed"
        Lamp1 (100,50 30x30), variable: MAIN.RoofControl.roofs[1].motors[1].opened, style: Lamp-Lamp1-Green
        Lamp1 (150,50 30x30), variable: MAIN.RoofControl.roofs[1].motors[1].closed, style: Lamp-Lamp1-Green
        Lamp1 (100,90 30x30), variable: MAIN.RoofControl.roofs[1].motors[2].opened, style: Lamp-Lamp1-Green
        Lamp1 (150,90 30x30), variable: MAIN.RoofControl.roofs[1].motors[2].closed, style: Lamp-Lamp1-Green
        Label (180,10 71x30), "Moving"
        Lamp1 (200,50 30x30), variable: MAIN.RoofControl.roofs[1].motors[1].moving, style: Lamp-Lamp1-Green
        Lamp1 (200,90 30x30), variable: MAIN.RoofControl.roofs[1].motors[2].moving, style: Lamp-Lamp1-Green
        Label (310,10 71x30), "Position"
        Textfield (350,50 41x30), "%.0f %", text variable: MAIN.RoofControl.roofs[1].motors[1].percent_open, input disabled if: TRUE
        Textfield (300,90 51x30), "%d", text variable: MAIN.RoofControl.roofs[1].motors[2].position, input disabled if: TRUE
        Label (400,10 71x30), "Speed"
        Textfield (400,50 71x30), "%.2f", text variable: MAIN.RoofControl.roofs[1].motors[1].speed, input disabled if: TRUE
        Textfield (400,90 71x30), "%.2f", text variable: MAIN.RoofControl.roofs[1].motors[2].speed, input disabled if: TRUE
        Label (480,10 71x30), "Open"
        PushSwitch (500,50 30x30), variable: MAIN.RoofControl.open_roof[1], behaviour: TAP, style: Switch-PushSwitch-Gray
        PushSwitch (550,50 30x30), variable: MAIN.RoofControl.close_roof[1], behaviour: TAP, style: Switch-PushSwitch-Gray
        Label (530,10 71x30), "Close"
        Label (590,10 51x30), "Stop"
        PushSwitch (600,50 30x30), variable: MAIN.RoofControl.stop_roof[1], behaviour: TAP, style: Switch-PushSwitch-Gray
        Lamp1 (500,90 30x30), variable: MAIN.RoofControl.roofs[1].sync_error, style: Lamp-Lamp1-Red
        Textfield (650,90 81x30), "%s", text variable: MAIN.RoofControl.roofs[1].state, input disabled if: TRUE
        Textfield (300,50 51x30), "%d", text variable: MAIN.RoofControl.roofs[1].motors[1].position, input disabled if: TRUE
        Textfield (350,90 41x30), "%.0f %", text variable: MAIN.RoofControl.roofs[1].motors[2].percent_open, input disabled if: TRUE
        Label (240,10 51x41), "Drive Error"
        Lamp1 (550,90 30x30), variable: MAIN.RoofControl.roofs[1].direction_error, style: Lamp-Lamp1-Red
        Label (490,120 51x41), "Sync error"
        Label (530,120 71x41), "Direction error"
        Label (640,10 51x30), "Reset"
        Lamp1 (250,50 30x30), variable: MAIN.RoofControl.roofs[1].motors[1].error, style: Lamp-Lamp1-Red
        Lamp1 (250,90 30x30), variable: MAIN.RoofControl.roofs[1].motors[2].error, style: Lamp-Lamp1-Red
        PushSwitch (750,50 30x30), variable: MAIN.RoofControl.roofs[1].slow_open, behaviour: TAP, style: Switch-PushSwitch-Red
        Label (740,10 51x31), "Slow open"
        Label (740,130 51x30), "Slow close"
        PushSwitch (750,230 30x30), variable: MAIN.RoofControl.stop_roof[1], behaviour: TAP, style: Switch-PushSwitch-Gray
        Label (690,10 51x31), "Zero counter"
        Lamp1 (600,90 30x30), variable: MAIN.RoofControl.roofs[1].limit_error, style: Lamp-Lamp1-Red
        Label (590,120 51x41), "Limit error"
    GroupBox (10,190 801x181), "Roof #2"
        Label (10,50 71x30), "Motor #1"
        Label (10,90 71x30), "Motor #2"
        Label (80,10 71x30), "Open"
        Label (130,10 71x30), "Closed"
        Lamp1 (100,50 30x30), variable: MAIN.RoofControl.roofs[2].motors[1].opened, style: Lamp-Lamp1-Green
        Lamp1 (150,50 30x30), variable: MAIN.RoofControl.roofs[2].motors[1].closed, style: Lamp-Lamp1-Green
        Lamp1 (100,90 30x30), variable: MAIN.RoofControl.roofs[2].motors[2].opened, style: Lamp-Lamp1-Green
        Lamp1 (150,90 30x30), variable: MAIN.RoofControl.roofs[2].motors[2].closed, style: Lamp-Lamp1-Green
        Label (180,10 71x30), "Moving"
        Lamp1 (200,50 30x30), variable: MAIN.RoofControl.roofs[2].motors[1].moving, style: Lamp-Lamp1-Green
        Lamp1 (200,90 30x30), variable: MAIN.RoofControl.roofs[2].motors[2].moving, style: Lamp-Lamp1-Green
        Label (310,10 71x30), "Position"
        Textfield (300,50 51x30), "%d", text variable: MAIN.RoofControl.roofs[2].motors[1].position, input disabled if: TRUE
        Textfield (300,90 51x30), "%d", text variable: MAIN.RoofControl.roofs[2].motors[2].position, input disabled if: TRUE
        Label (400,10 71x30), "Speed"
        Textfield (400,50 71x30), "%.2f", text variable: MAIN.RoofControl.roofs[2].motors[1].speed, input disabled if: TRUE
        Textfield (400,90 71x30), "%.2f", text variable: MAIN.RoofControl.roofs[2].motors[2].speed, input disabled if: TRUE
        Label (480,10 71x30), "Open"
        PushSwitch (500,50 30x30), variable: MAIN.RoofControl.open_roof[2], behaviour: TAP, style: Switch-PushSwitch-Gray
        PushSwitch (550,50 30x30), variable: MAIN.RoofControl.close_roof[2], behaviour: TAP, style: Switch-PushSwitch-Gray
        Label (530,10 71x30), "Close"
        Label (590,10 51x30), "Stop"
        PushSwitch (600,50 30x30), variable: MAIN.RoofControl.stop_roof[2], behaviour: TAP, style: Switch-PushSwitch-Gray
        Lamp1 (500,90 30x30), variable: MAIN.RoofControl.roofs[2].sync_error, style: Lamp-Lamp1-Red
        Textfield (650,90 81x30), "%s", text variable: MAIN.RoofControl.roofs[2].state, input disabled if: TRUE
        Textfield (350,50 41x30), "%.0f %", text variable: MAIN.RoofControl.roofs[2].motors[1].percent_open, input disabled if: TRUE
        Textfield (350,90 41x30), "%.0f %", text variable: MAIN.RoofControl.roofs[2].motors[2].percent_open, input disabled if: TRUE
        Label (240,10 51x41), "Drive Error"
        Label (490,130 51x41), "Sync error"
        Label (530,130 71x41), "Direction error"
        Lamp1 (550,90 30x30), variable: MAIN.RoofControl.roofs[2].direction_error, style: Lamp-Lamp1-Red
        Lamp1 (250,90 30x30), variable: MAIN.RoofControl.roofs[2].motors[2].error, style: Lamp-Lamp1-Red
        Lamp1 (250,50 30x30), variable: MAIN.RoofControl.roofs[2].motors[1].error, style: Lamp-Lamp1-Red
        PushSwitch (750,50 30x30), variable: MAIN.RoofControl.roofs[2].slow_open, behaviour: TAP, style: Switch-PushSwitch-Red
        PushSwitch (750,90 30x30), variable: MAIN.RoofControl.stop_roof[1], behaviour: TAP, style: Switch-PushSwitch-Gray
        PushSwitch (750,-90 30x30), variable: MAIN.RoofControl.stop_roof[1], behaviour: TAP, style: Switch-PushSwitch-Gray
        Label (740,130 51x30), "Slow close"
        Label (690,10 51x31), "Zero counter"
        Lamp1 (600,90 30x30), variable: MAIN.RoofControl.roofs[2].limit_error, style: Lamp-Lamp1-Red
        Label (590,130 51x41), "Limit error"
    GroupBox (820,10 151x361), "Roof"
        Label (70,150 71x30), "Open"
        PushSwitch (20,150 30x30), variable: MAIN.RoofControl.open_roofs, behaviour: TAP, style: Switch-PushSwitch-Gray
        PushSwitch (20,190 30x30), variable: MAIN.RoofControl.close_roofs, behaviour: TAP, style: Switch-PushSwitch-Gray
        Label (70,190 71x30), "Close"
        Label (70,250 71x30), "Stop"
        PushSwitch (20,250 30x30), variable: MAIN.RoofControl.stop_roofs, behaviour: TAP, style: Switch-PushSwitch-Red
        Label (70,90 71x30), "Automatic"
        Lamp1 (20,90 30x30), variable: MAIN.RoofControl.automatic, style: Lamp-Lamp1-Yellow
        Label (70,310 71x30), "Reset"
        PushSwitch (20,310 30x30), variable: MAIN.RoofControl.reset_roofs, behaviour: TAP, style: Switch-PushSwitch-Gray
        Textfield (20,50 111x30), "%s", text variable: MAIN.RoofControl.roofs[1].state, input disabled if: TRUE
    PushSwitch (660,60 30x30), variable: MAIN.RoofControl.reset_roof[1], behaviour: TAP, style: Switch-PushSwitch-Gray
    Label (650,200 51x30), "Reset"
    PushSwitch (660,240 30x30), variable: MAIN.RoofControl.reset_roof[2], behaviour: TAP, style: Switch-PushSwitch-Gray
    PushSwitch (710,60 30x30), variable: MAIN.RoofControl.roofs[1].zero_counter, behaviour: TAP, style: Switch-PushSwitch-Yellow
    Label (750,200 51x31), "Slow open"
    PushSwitch (710,240 30x30), variable: MAIN.RoofControl.roofs[2].zero_counter, behaviour: TAP, style: Switch-PushSwitch-Yellow
    PushSwitch (760,280 30x30), variable: MAIN.RoofControl.roofs[2].slow_close, behaviour: TAP, style: Switch-PushSwitch-Red
    PushSwitch (760,100 30x30), variable: MAIN.RoofControl.roofs[1].slow_close, behaviour: TAP, style: Switch-PushSwitch-Red
END_VISUALIZATION
